LIN {X 0,Y 514.974,Z 940.438,A -85,B 0,C 180,E1 22806.113,E2 22806.113} C_VEL
LIN {X 0,Y 511.888,Z 958.496,A -85,B 0,C 180,E1 22805.05,E2 22805.05} C_VEL
LIN {X 0,Y 508.208,Z 978.384,A -85,B 0,C 180,E1 22803.67,E2 22803.67} C_VEL
LIN {X 0,Y 504.574,Z 996.273,A -85,B 0,C 180,E1 22802.202,E2 22802.202} C_VEL
LIN {X 0,Y 500.609,Z 1014.935,A -85,B 0,C 180,E1 22800.42,E2 22800.42} C_VEL
LIN {X 0,Y 500.137,Z 1017.069,A -85,B 0,C 180,E1 22800.192,E2 22800.192} C_VEL
LIN {X 0,Y 498.01,Z 1022.89,A -85,B 0,C 180,E1 22799.633,E2 22799.633} C_VEL
LIN {X 0,Y 489.476,Z 1037.041,A -85,B 0,C 180,E1 22798.306,E2 22798.306} C_VEL
LIN {X 0,Y 487.395,Z 1042.192,A -85,B 0,C 180,E1 22797.684,E2 22797.684} C_VEL
LIN {X 0,Y 483.645,Z 1058.175,A -85,B 0,C 180,E1 22795.338,E2 22795.338} C_VEL
LIN {X 0,Y 480.612,Z 1071.674,A -85,B 0,C 180,E1 22793.025,E2 22793.025} C_VEL
LIN {X 0,Y 477.995,Z 1083.738,A -85,B 0,C 180,E1 22790.575,E2 22790.575} C_VEL
LIN {X 0,Y 475.867,Z 1094.639,A -85,B 0,C 180,E1 22787.992,E2 22787.992} C_VEL
LIN {X 0,Y 474.237,Z 1103.992,A -85,B 0,C 180,E1 22785.281,E2 22785.281} C_VEL
LIN {X 0,Y 473.115,Z 1112.013,A -85,B 0,C 180,E1 22782.449,E2 22782.449} C_VEL
LIN {X 0,Y 472.494,Z 1117.73,A -85,B 0,C 180,E1 22779.87,E2 22779.87} C_VEL
LIN {X 0,Y 472.112,Z 1122.616,A -85,B 0,C 180,E1 22776.934,E2 22776.934} C_VEL
LIN {X 0,Y 471.982,Z 1125.43,A -85,B 0,C 180,E1 22774.374,E2 22774.374} C_VEL
LIN {X 0,Y 471.935,Z 1127.131,A -85,B 0,C 180,E1 22771.457,E2 22771.457} C_VEL
LIN {X 0,Y 471.943,Z 1127.212,A -85,B 0,C 180,E1 22768.907,E2 22768.907} C_VEL
LIN {X 0,Y 471.968,Z 1125.953,A -85,B 0,C 180,E1 22766.113,E2 22766.113} C_VEL
LIN {X 0,Y 472.089,Z 1123.143,A -85,B 0,C 180,E1 22763.39,E2 22763.39} C_VEL
LIN {X 0,Y 472.386,Z 1118.901,A -85,B 0,C 180,E1 22760.62,E2 22760.62} C_VEL
LIN {X 0,Y 472.973,Z 1113.117,A -85,B 0,C 180,E1 22757.919,E2 22757.919} C_VEL
LIN {X 0,Y 474.03,Z 1105.47,A -85,B 0,C 180,E1 22755.088,E2 22755.088} C_VEL
LIN {X 0,Y 475.474,Z 1096.754,A -85,B 0,C 180,E1 22752.499,E2 22752.499} C_VEL
LIN {X 0,Y 477.693,Z 1085.268,A -85,B 0,C 180,E1 22749.668,E2 22749.668} C_VEL
LIN {X 0,Y 480.112,Z 1073.916,A -85,B 0,C 180,E1 22747.31,E2 22747.31} C_VEL
LIN {X 0,Y 483.191,Z 1060.24,A -85,B 0,C 180,E1 22744.899,E2 22744.899} C_VEL
LIN {X 0,Y 486.557,Z 1045.907,A -85,B 0,C 180,E1 22742.724,E2 22742.724} C_VEL
LIN {X 0,Y 490.327,Z 1029.688,A -85,B 0,C 180,E1 22740.631,E2 22740.631} C_VEL
LIN {X 0,Y 494.255,Z 1012.751,A -85,B 0,C 180,E1 22738.738,E2 22738.738} C_VEL
LIN {X 0,Y 498.243,Z 994.544,A -85,B 0,C 180,E1 22737.02,E2 22737.02} C_VEL
LIN {X 0,Y 502.323,Z 975.012,A -85,B 0,C 180,E1 22735.437,E2 22735.437} C_VEL
LIN {X 0,Y 505.787,Z 956.671,A -85,B 0,C 180,E1 22734.185,E2 22734.185} C_VEL
LIN {X 0,Y 509.321,Z 936.541,A -85,B 0,C 180,E1 22733.014,E2 22733.014} C_VEL
LIN {X 0,Y 512.447,Z 915.409,A -85,B 0,C 180,E1 22732.011,E2 22732.011} C_VEL
LIN {X 0,Y 515.345,Z 892.845,A -85,B 0,C 180,E1 22731.144,E2 22731.144} C_VEL
LIN {X 0,Y 517.532,Z 870.869,A -85,B 0,C 180,E1 22730.501,E2 22730.501} C_VEL
LIN {X 0,Y 519.328,Z 846.322,A -85,B 0,C 180,E1 22729.983,E2 22729.983} C_VEL
LIN {X 0,Y 527.013,Z 617.451,A -85,B 0,C 180,E1 22726.684,E2 22726.684} C_VEL
LIN {X 0,Y 529.08,Z 555.866,A -85,B 0,C 180,E1 22725.782,E2 22725.782} C_VEL
LIN {X 0,Y 524.909,Z 533.069,A -85,B 0,C 180,E1 22724.874,E2 22724.874} C_VEL
LIN {X 0,Y 515.36,Z 516.714,A -85,B 0,C 180,E1 22723.399,E2 22723.399} C_VEL
LIN {X 0,Y 504.426,Z 499.31,A -85,B 0,C 180,E1 22721.61,E2 22721.61} C_VEL
LIN {X 0,Y 497.117,Z 487.981,A -85,B 0,C 180,E1 22720.29,E2 22720.29} C_VEL
LIN {X 0,Y 491.248,Z 474.305,A -85,B 0,C 180,E1 22717.635,E2 22717.635} C_VEL
LIN {X 0,Y 486.199,Z 463.352,A -85,B 0,C 180,E1 22715.269,E2 22715.269} C_VEL
LIN {X 0,Y 482.496,Z 455.619,A -85,B 0,C 180,E1 22713.452,E2 22713.452} C_VEL
LIN {X 0,Y 480.184,Z 450.949,A -85,B 0,C 180,E1 22712.283,E2 22712.283} C_VEL
LIN {X 0,Y 478.108,Z 446.81,A -85,B 0,C 180,E1 22711.2,E2 22711.2} C_VEL
LIN {X 0,Y 475.909,Z 442.427,A -85,B 0,C 180,E1 22710.003,E2 22710.003} C_VEL
LIN {X 0,Y 474.193,Z 438.99,A -85,B 0,C 180,E1 22709.011,E2 22709.011} C_VEL
LIN {X 0,Y 474.091,Z 438.231,A -85,B 0,C 180,E1 22708.672,E2 22708.672} C_VEL
LIN {X 0,Y 474.033,Z 438.161,A -85,B 0,C 180,E1 22705.086,E2 22705.086} C_VEL
LIN {X 0,Y 474.022,Z 438.165,A -85,B 0,C 180,E1 22701.663,E2 22701.663} C_VEL
LIN {X 0,Y 474.067,Z 438.17,A -85,B 0,C 180,E1 22698.189,E2 22698.189} C_VEL
LIN {X 0,Y 474.07,Z 438.181,A -85,B 0,C 180,E1 22694.661,E2 22694.661} C_VEL
LIN {X 0,Y 474.036,Z 438.17,A -85,B 0,C 180,E1 22691.19,E2 22691.19} C_VEL
LIN {X 0,Y 474.042,Z 438.155,A -85,B 0,C 180,E1 22687.514,E2 22687.514} C_VEL
LIN {X 0,Y 474.09,Z 438.146,A -85,B 0,C 180,E1 22684.112,E2 22684.112} C_VEL
LIN {X 0,Y 474.07,Z 438.166,A -85,B 0,C 180,E1 22680.604,E2 22680.604} C_VEL
LIN {X 0,Y 474.053,Z 438.18,A -85,B 0,C 180,E1 22677.098,E2 22677.098} C_VEL
LIN {X 0,Y 474.066,Z 438.161,A -85,B 0,C 180,E1 22673.46,E2 22673.46} C_VEL
LIN {X 0,Y 474.105,Z 438.145,A -85,B 0,C 180,E1 22670.034,E2 22670.034} C_VEL
LIN {X 0,Y 474.076,Z 438.152,A -85,B 0,C 180,E1 22666.461,E2 22666.461} C_VEL
LIN {X 0,Y 474.067,Z 438.164,A -85,B 0,C 180,E1 22662.952,E2 22662.952} C_VEL
LIN {X 0,Y 474.094,Z 438.17,A -85,B 0,C 180,E1 22659.377,E2 22659.377} C_VEL
LIN {X 0,Y 474.117,Z 438.173,A -85,B 0,C 180,E1 22655.849,E2 22655.849} C_VEL
LIN {X 0,Y 474.103,Z 438.234,A -85,B 0,C 180,E1 22652.219,E2 22652.219} C_VEL
LIN {X 0,Y 474.211,Z 438.738,A -85,B 0,C 180,E1 22651.884,E2 22651.884} C_VEL
LIN {X 0,Y 476.008,Z 442.457,A -85,B 0,C 180,E1 22650.834,E2 22650.834} C_VEL
LIN {X 0,Y 479.297,Z 448.858,A -85,B 0,C 180,E1 22649.123,E2 22649.123} C_VEL
LIN {X 0,Y 481.852,Z 453.929,A -85,B 0,C 180,E1 22647.849,E2 22647.849} C_VEL
LIN {X 0,Y 485.845,Z 461.926,A -85,B 0,C 180,E1 22645.959,E2 22645.959} C_VEL
LIN {X 0,Y 487.43,Z 464.88,A -85,B 0,C 180,E1 22645.373,E2 22645.373} C_VEL
LIN {X 0,Y 499.532,Z 481.118,A -85,B 0,C 180,E1 22643.148,E2 22643.148} C_VEL
LIN {X 0,Y 512.045,Z 499.258,A -85,B 0,C 180,E1 22641.039,E2 22641.039} C_VEL
LIN {X 0,Y 523.907,Z 517.752,A -85,B 0,C 180,E1 22639.181,E2 22639.181} C_VEL
LIN {X 0,Y 531.983,Z 531.498,A -85,B 0,C 180,E1 22637.975,E2 22637.975} C_VEL
LIN {X 0,Y 522.698,Z 768.418,A -85,B 0,C 180,E1 22634.376,E2 22634.376} C_VEL
LIN {X 0,Y 519.654,Z 844.715,A -85,B 0,C 180,E1 22633.19,E2 22633.19} C_VEL
LIN {X 0,Y 517.66,Z 869.839,A -85,B 0,C 180,E1 22632.628,E2 22632.628} C_VEL
LIN {X 0,Y 515.301,Z 892.72,A -85,B 0,C 180,E1 22631.945,E2 22631.945} C_VEL
LIN {X 0,Y 512.362,Z 915.91,A -85,B 0,C 180,E1 22631.048,E2 22631.048} C_VEL
LIN {X 0,Y 509.382,Z 936.467,A -85,B 0,C 180,E1 22630.08,E2 22630.08} C_VEL
LIN {X 0,Y 505.522,Z 959.82,A -85,B 0,C 180,E1 22628.757,E2 22628.757} C_VEL
LIN {X 0,Y 502.089,Z 978.916,A -85,B 0,C 180,E1 22627.474,E2 22627.474} C_VEL
LIN {X 0,Y 497.871,Z 1000.724,A -85,B 0,C 180,E1 22625.763,E2 22625.763} C_VEL
LIN {X 0,Y 494.305,Z 1018.112,A -85,B 0,C 180,E1 22624.174,E2 22624.174} C_VEL
LIN {X 0,Y 490.354,Z 1037.041,A -85,B 0,C 180,E1 22622.195,E2 22622.195} C_VEL
LIN {X 0,Y 486.762,Z 1053.913,A -85,B 0,C 180,E1 22620.139,E2 22620.139} C_VEL
LIN {X 0,Y 483.383,Z 1070.255,A -85,B 0,C 180,E1 22617.871,E2 22617.871} C_VEL
LIN {X 0,Y 480.434,Z 1084.78,A -85,B 0,C 180,E1 22615.519,E2 22615.519} C_VEL
LIN {X 0,Y 477.873,Z 1098.534,A -85,B 0,C 180,E1 22612.979,E2 22612.979} C_VEL
LIN {X 0,Y 475.763,Z 1110.817,A -85,B 0,C 180,E1 22610.29,E2 22610.29} C_VEL
LIN {X 0,Y 474.199,Z 1121.612,A -85,B 0,C 180,E1 22607.549,E2 22607.549} C_VEL
LIN {X 0,Y 473.122,Z 1130.443,A -85,B 0,C 180,E1 22604.816,E2 22604.816} C_VEL
LIN {X 0,Y 472.485,Z 1137.458,A -85,B 0,C 180,E1 22602.218,E2 22602.218} C_VEL
LIN {X 0,Y 472.088,Z 1143.705,A -85,B 0,C 180,E1 22599.249,E2 22599.249} C_VEL
LIN {X 0,Y 471.972,Z 1147.524,A -85,B 0,C 180,E1 22596.814,E2 22596.814} C_VEL
LIN {X 0,Y 471.934,Z 1150.574,A -85,B 0,C 180,E1 22594.009,E2 22594.009} C_VEL
LIN {X 0,Y 471.933,Z 1151.919,A -85,B 0,C 180,E1 22591.214,E2 22591.214} C_VEL
LIN {X 0,Y 471.93,Z 1151.942,A -85,B 0,C 180,E1 22588.907,E2 22588.907} C_VEL
LIN {X 0,Y 471.931,Z 1150.773,A -85,B 0,C 180,E1 22586.307,E2 22586.307} C_VEL
LIN {X 0,Y 471.964,Z 1147.852,A -85,B 0,C 180,E1 22583.431,E2 22583.431} C_VEL
LIN {X 0,Y 472.068,Z 1144.104,A -85,B 0,C 180,E1 22580.982,E2 22580.982} C_VEL
LIN {X 0,Y 472.41,Z 1138.385,A -85,B 0,C 180,E1 22578.152,E2 22578.152} C_VEL
LIN {X 0,Y 473.04,Z 1131.162,A -85,B 0,C 180,E1 22575.431,E2 22575.431} C_VEL
LIN {X 0,Y 473.962,Z 1123.279,A -85,B 0,C 180,E1 22572.948,E2 22572.948} C_VEL
LIN {X 0,Y 475.544,Z 1112.173,A -85,B 0,C 180,E1 22570.031,E2 22570.031} C_VEL
LIN {X 0,Y 477.369,Z 1101.223,A -85,B 0,C 180,E1 22567.591,E2 22567.591} C_VEL
LIN {X 0,Y 480.025,Z 1086.91,A -85,B 0,C 180,E1 22564.854,E2 22564.854} C_VEL
LIN {X 0,Y 482.698,Z 1073.379,A -85,B 0,C 180,E1 22562.621,E2 22562.621} C_VEL
LIN {X 0,Y 486.389,Z 1055.696,A -85,B 0,C 180,E1 22560.098,E2 22560.098} C_VEL
LIN {X 0,Y 489.701,Z 1039.918,A -85,B 0,C 180,E1 22558.147,E2 22558.147} C_VEL
LIN {X 0,Y 493.993,Z 1019.506,A -85,B 0,C 180,E1 22555.967,E2 22555.967} C_VEL
LIN {X 0,Y 497.576,Z 1001.995,A -85,B 0,C 180,E1 22554.355,E2 22554.355} C_VEL
LIN {X 0,Y 501.927,Z 979.629,A -85,B 0,C 180,E1 22552.584,E2 22552.584} C_VEL
LIN {X 0,Y 505.349,Z 960.615,A -85,B 0,C 180,E1 22551.3,E2 22551.3} C_VEL
LIN {X 0,Y 509.174,Z 937.611,A -85,B 0,C 180,E1 22549.984,E2 22549.984} C_VEL
LIN {X 0,Y 512.166,Z 917.021,A -85,B 0,C 180,E1 22549.007,E2 22549.007} C_VEL
LIN {X 0,Y 515.216,Z 893.121,A -85,B 0,C 180,E1 22548.075,E2 22548.075} C_VEL
LIN {X 0,Y 517.586,Z 870.113,A -85,B 0,C 180,E1 22547.385,E2 22547.385} C_VEL
LIN {X 0,Y 519.577,Z 845.22,A -85,B 0,C 180,E1 22546.825,E2 22546.825} C_VEL
LIN {X 0,Y 522.328,Z 776.987,A -85,B 0,C 180,E1 22545.762,E2 22545.762} C_VEL
LIN {X 0,Y 531.499,Z 541.74,A -85,B 0,C 180,E1 22542.186,E2 22542.186} C_VEL
LIN {X 0,Y 531.834,Z 531.038,A -85,B 0,C 180,E1 22542.014,E2 22542.014} C_VEL
LIN {X 0,Y 519.165,Z 510.17,A -85,B 0,C 180,E1 22540.108,E2 22540.108} C_VEL
LIN {X 0,Y 506.446,Z 491.019,A -85,B 0,C 180,E1 22538.06,E2 22538.06} C_VEL
LIN {X 0,Y 494.73,Z 474.66,A -85,B 0,C 180,E1 22536.025,E2 22536.025} C_VEL
LIN {X 0,Y 486.873,Z 464.103,A -85,B 0,C 180,E1 22534.529,E2 22534.529} C_VEL
LIN {X 0,Y 482.962,Z 456.048,A -85,B 0,C 180,E1 22532.708,E2 22532.708} C_VEL
LIN {X 0,Y 480.419,Z 451.159,A -85,B 0,C 180,E1 22531.494,E2 22531.494} C_VEL
LIN {X 0,Y 478.261,Z 446.86,A -85,B 0,C 180,E1 22530.394,E2 22530.394} C_VEL
LIN {X 0,Y 475.915,Z 442.341,A -85,B 0,C 180,E1 22529.172,E2 22529.172} C_VEL
LIN {X 0,Y 474.23,Z 438.807,A -85,B 0,C 180,E1 22528.183,E2 22528.183} C_VEL
LIN {X 0,Y 474.102,Z 438.209,A -85,B 0,C 180,E1 22527.781,E2 22527.781} C_VEL
LIN {X 0,Y 474.118,Z 438.172,A -85,B 0,C 180,E1 22524.151,E2 22524.151} C_VEL
LIN {X 0,Y 474.103,Z 438.171,A -85,B 0,C 180,E1 22520.543,E2 22520.543} C_VEL
LIN {X 0,Y 474.069,Z 438.163,A -85,B 0,C 180,E1 22517.048,E2 22517.048} C_VEL
LIN {X 0,Y 474.07,Z 438.154,A -85,B 0,C 180,E1 22513.415,E2 22513.415} C_VEL
LIN {X 0,Y 474.108,Z 438.145,A -85,B 0,C 180,E1 22509.959,E2 22509.959} C_VEL
LIN {X 0,Y 474.069,Z 438.161,A -85,B 0,C 180,E1 22506.54,E2 22506.54} C_VEL
LIN {X 0,Y 474.055,Z 438.18,A -85,B 0,C 180,E1 22502.902,E2 22502.902} C_VEL
LIN {X 0,Y 474.075,Z 438.165,A -85,B 0,C 180,E1 22499.396,E2 22499.396} C_VEL
LIN {X 0,Y 474.092,Z 438.145,A -85,B 0,C 180,E1 22495.888,E2 22495.888} C_VEL
LIN {X 0,Y 474.047,Z 438.155,A -85,B 0,C 180,E1 22492.463,E2 22492.463} C_VEL
LIN {X 0,Y 474.043,Z 438.171,A -85,B 0,C 180,E1 22488.81,E2 22488.81} C_VEL
LIN {X 0,Y 474.079,Z 438.18,A -85,B 0,C 180,E1 22485.339,E2 22485.339} C_VEL
LIN {X 0,Y 474.069,Z 438.167,A -85,B 0,C 180,E1 22481.811,E2 22481.811} C_VEL
LIN {X 0,Y 474.027,Z 438.163,A -85,B 0,C 180,E1 22478.337,E2 22478.337} C_VEL
LIN {X 0,Y 474.035,Z 438.161,A -85,B 0,C 180,E1 22474.781,E2 22474.781} C_VEL
LIN {X 0,Y 474.087,Z 438.218,A -85,B 0,C 180,E1 22471.257,E2 22471.257} C_VEL
LIN {X 0,Y 474.125,Z 438.668,A -85,B 0,C 180,E1 22470.932,E2 22470.932} C_VEL
LIN {X 0,Y 475.635,Z 442.084,A -85,B 0,C 180,E1 22469.978,E2 22469.978} C_VEL
LIN {X 0,Y 476.655,Z 443.662,A -85,B 0,C 180,E1 22469.492,E2 22469.492} C_VEL
LIN {X 0,Y 478.533,Z 447.391,A -85,B 0,C 180,E1 22468.487,E2 22468.487} C_VEL
LIN {X 0,Y 481.515,Z 453.713,A -85,B 0,C 180,E1 22466.898,E2 22466.898} C_VEL
LIN {X 0,Y 485.309,Z 461.34,A -85,B 0,C 180,E1 22465.056,E2 22465.056} C_VEL
LIN {X 0,Y 491.281,Z 474.454,A -85,B 0,C 180,E1 22462.221,E2 22462.221} C_VEL
LIN {X 0,Y 497.06,Z 487.845,A -85,B 0,C 180,E1 22459.628,E2 22459.628} C_VEL
LIN {X 0,Y 499.745,Z 492.282,A -85,B 0,C 180,E1 22459.079,E2 22459.079} C_VEL
LIN {X 0,Y 510.188,Z 508.318,A -85,B 0,C 180,E1 22457.323,E2 22457.323} C_VEL
LIN {X 0,Y 522.638,Z 529.103,A -85,B 0,C 180,E1 22455.363,E2 22455.363} C_VEL
LIN {X 0,Y 525.199,Z 534.086,A -85,B 0,C 180,E1 22454.967,E2 22454.967} C_VEL
LIN {X 0,Y 529.111,Z 557.421,A -85,B 0,C 180,E1 22454.081,E2 22454.081} C_VEL
LIN {X 0,Y 520.357,Z 817.692,A -85,B 0,C 180,E1 22450.349,E2 22450.349} C_VEL
LIN {X 0,Y 518.943,Z 852.159,A -85,B 0,C 180,E1 22449.818,E2 22449.818} C_VEL
LIN {X 0,Y 517.154,Z 874.464,A -85,B 0,C 180,E1 22449.31,E2 22449.31} C_VEL
LIN {X 0,Y 514.604,Z 898.665,A -85,B 0,C 180,E1 22448.552,E2 22448.552} C_VEL
LIN {X 0,Y 511.976,Z 918.576,A -85,B 0,C 180,E1 22447.754,E2 22447.754} C_VEL
LIN {X 0,Y 508.507,Z 941.041,A -85,B 0,C 180,E1 22446.64,E2 22446.64} C_VEL
LIN {X 0,Y 505.173,Z 959.846,A -85,B 0,C 180,E1 22445.516,E2 22445.516} C_VEL
LIN {X 0,Y 501.125,Z 980.634,A -85,B 0,C 180,E1 22444.034,E2 22444.034} C_VEL
LIN {X 0,Y 497.359,Z 998.511,A -85,B 0,C 180,E1 22442.533,E2 22442.533} C_VEL
LIN {X 0,Y 493.253,Z 1016.9,A -85,B 0,C 180,E1 22440.72,E2 22440.72} C_VEL
LIN {X 0,Y 489.571,Z 1032.936,A -85,B 0,C 180,E1 22438.883,E2 22438.883} C_VEL
LIN {X 0,Y 487.395,Z 1042.192,A -85,B 0,C 180,E1 22437.684,E2 22437.684} C_VEL
LIN {X 0,Y 485.339,Z 1047.343,A -85,B 0,C 180,E1 22437.042,E2 22437.042} C_VEL
LIN {X 0,Y 476.907,Z 1060.015,A -85,B 0,C 180,E1 22435.473,E2 22435.473} C_VEL
LIN {X 0,Y 474.868,Z 1064.523,A -85,B 0,C 180,E1 22434.753,E2 22434.753} C_VEL
LIN {X 0,Y 471.929,Z 1076.945,A -85,B 0,C 180,E1 22432.419,E2 22432.419} C_VEL
LIN {X 0,Y 469.326,Z 1088.898,A -85,B 0,C 180,E1 22429.801,E2 22429.801} C_VEL
LIN {X 0,Y 467.35,Z 1098.886,A -85,B 0,C 180,E1 22427.173,E2 22427.173} C_VEL
LIN {X 0,Y 465.767,Z 1108.276,A -85,B 0,C 180,E1 22424.166,E2 22424.166} C_VEL
LIN {X 0,Y 464.847,Z 1115.168,A -85,B 0,C 180,E1 22421.414,E2 22421.414} C_VEL
LIN {X 0,Y 464.295,Z 1120.599,A -85,B 0,C 180,E1 22418.546,E2 22418.546} C_VEL
LIN {X 0,Y 464.05,Z 1124.214,A -85,B 0,C 180,E1 22415.937,E2 22415.937} C_VEL
LIN {X 0,Y 463.959,Z 1126.617,A -85,B 0,C 180,E1 22413.089,E2 22413.089} C_VEL
LIN {X 0,Y 463.943,Z 1127.492,A -85,B 0,C 180,E1 22410.617,E2 22410.617} C_VEL
LIN {X 0,Y 463.948,Z 1127.06,A -85,B 0,C 180,E1 22407.653,E2 22407.653} C_VEL
LIN {X 0,Y 464,Z 1125.29,A -85,B 0,C 180,E1 22405.055,E2 22405.055} C_VEL
LIN {X 0,Y 464.2,Z 1121.946,A -85,B 0,C 180,E1 22402.201,E2 22402.201} C_VEL
LIN {X 0,Y 464.608,Z 1117.157,A -85,B 0,C 180,E1 22399.459,E2 22399.459} C_VEL
LIN {X 0,Y 465.431,Z 1110.588,A -85,B 0,C 180,E1 22396.584,E2 22396.584} C_VEL
LIN {X 0,Y 466.624,Z 1102.952,A -85,B 0,C 180,E1 22393.953,E2 22393.953} C_VEL
LIN {X 0,Y 468.533,Z 1092.768,A -85,B 0,C 180,E1 22391.072,E2 22391.072} C_VEL
LIN {X 0,Y 470.779,Z 1082.168,A -85,B 0,C 180,E1 22388.573,E2 22388.573} C_VEL
LIN {X 0,Y 473.781,Z 1069.027,A -85,B 0,C 180,E1 22385.963,E2 22385.963} C_VEL
LIN {X 0,Y 477.129,Z 1055.239,A -85,B 0,C 180,E1 22383.623,E2 22383.623} C_VEL
LIN {X 0,Y 480.825,Z 1039.945,A -85,B 0,C 180,E1 22381.426,E2 22381.426} C_VEL
LIN {X 0,Y 484.873,Z 1023.467,A -85,B 0,C 180,E1 22379.379,E2 22379.379} C_VEL
LIN {X 0,Y 488.838,Z 1006.54,A -85,B 0,C 180,E1 22377.594,E2 22377.594} C_VEL
LIN {X 0,Y 493.061,Z 987.865,A -85,B 0,C 180,E1 22375.894,E2 22375.894} C_VEL
LIN {X 0,Y 496.966,Z 969.009,A -85,B 0,C 180,E1 22374.446,E2 22374.446} C_VEL
LIN {X 0,Y 501.016,Z 947.927,A -85,B 0,C 180,E1 22373.079,E2 22373.079} C_VEL
LIN {X 0,Y 504.386,Z 927.99,A -85,B 0,C 180,E1 22372.009,E2 22372.009} C_VEL
LIN {X 0,Y 507.772,Z 904.722,A -85,B 0,C 180,E1 22370.991,E2 22370.991} C_VEL
LIN {X 0,Y 510.184,Z 884.575,A -85,B 0,C 180,E1 22370.295,E2 22370.295} C_VEL
LIN {X 0,Y 512.428,Z 860.395,A -85,B 0,C 180,E1 22369.663,E2 22369.663} C_VEL
LIN {X 0,Y 513.755,Z 838.487,A -85,B 0,C 180,E1 22369.26,E2 22369.26} C_VEL
LIN {X 0,Y 522.47,Z 588.071,A -85,B 0,C 180,E1 22365.635,E2 22365.635} C_VEL
LIN {X 0,Y 523.48,Z 557.529,A -85,B 0,C 180,E1 22365.174,E2 22365.174} C_VEL
LIN {X 0,Y 519.86,Z 537.391,A -85,B 0,C 180,E1 22364.359,E2 22364.359} C_VEL
LIN {X 0,Y 508.793,Z 518.402,A -85,B 0,C 180,E1 22362.592,E2 22362.592} C_VEL
LIN {X 0,Y 497.226,Z 500.156,A -85,B 0,C 180,E1 22360.62,E2 22360.62} C_VEL
LIN {X 0,Y 488.867,Z 487.482,A -85,B 0,C 180,E1 22359.047,E2 22359.047} C_VEL
LIN {X 0,Y 482.492,Z 473.005,A -85,B 0,C 180,E1 22356.054,E2 22356.054} C_VEL
LIN {X 0,Y 477.244,Z 461.72,A -85,B 0,C 180,E1 22353.437,E2 22353.437} C_VEL
LIN {X 0,Y 472.696,Z 452.61,A -85,B 0,C 180,E1 22351.073,E2 22351.073} C_VEL
LIN {X 0,Y 470.426,Z 448.145,A -85,B 0,C 180,E1 22349.826,E2 22349.826} C_VEL
LIN {X 0,Y 468.616,Z 444.219,A -85,B 0,C 180,E1 22348.722,E2 22348.722} C_VEL
LIN {X 0,Y 466.315,Z 440.328,A -85,B 0,C 180,E1 22347.453,E2 22347.453} C_VEL
LIN {X 0,Y 466.113,Z 439.268,A -85,B 0,C 180,E1 22347.051,E2 22347.051} C_VEL
LIN {X 0,Y 466.081,Z 439.159,A -85,B 0,C 180,E1 22343.518,E2 22343.518} C_VEL
LIN {X 0,Y 466.1,Z 439.151,A -85,B 0,C 180,E1 22339.943,E2 22339.943} C_VEL
LIN {X 0,Y 466.145,Z 439.138,A -85,B 0,C 180,E1 22336.448,E2 22336.448} C_VEL
LIN {X 0,Y 466.1,Z 439.144,A -85,B 0,C 180,E1 22333.018,E2 22333.018} C_VEL
LIN {X 0,Y 466.097,Z 439.154,A -85,B 0,C 180,E1 22329.383,E2 22329.383} C_VEL
LIN {X 0,Y 466.135,Z 439.167,A -85,B 0,C 180,E1 22325.91,E2 22325.91} C_VEL
LIN {X 0,Y 466.159,Z 439.15,A -85,B 0,C 180,E1 22322.213,E2 22322.213} C_VEL
LIN {X 0,Y 466.117,Z 439.138,A -85,B 0,C 180,E1 22318.771,E2 22318.771} C_VEL
LIN {X 0,Y 466.112,Z 439.142,A -85,B 0,C 180,E1 22315.201,E2 22315.201} C_VEL
LIN {X 0,Y 466.157,Z 439.157,A -85,B 0,C 180,E1 22311.737,E2 22311.737} C_VEL
LIN {X 0,Y 466.168,Z 439.163,A -85,B 0,C 180,E1 22308.117,E2 22308.117} C_VEL
LIN {X 0,Y 466.133,Z 439.151,A -85,B 0,C 180,E1 22304.574,E2 22304.574} C_VEL
LIN {X 0,Y 466.131,Z 439.143,A -85,B 0,C 180,E1 22300.971,E2 22300.971} C_VEL
LIN {X 0,Y 466.163,Z 439.137,A -85,B 0,C 180,E1 22297.422,E2 22297.422} C_VEL
LIN {X 0,Y 466.2,Z 439.306,A -85,B 0,C 180,E1 22293.704,E2 22293.704} C_VEL
LIN {X 0,Y 467.592,Z 442.857,A -85,B 0,C 180,E1 22292.629,E2 22292.629} C_VEL
LIN {X 0,Y 468.898,Z 444.787,A -85,B 0,C 180,E1 22291.986,E2 22291.986} C_VEL
LIN {X 0,Y 470.858,Z 448.554,A -85,B 0,C 180,E1 22290.903,E2 22290.903} C_VEL
LIN {X 0,Y 474.049,Z 455.088,A -85,B 0,C 180,E1 22289.166,E2 22289.166} C_VEL
LIN {X 0,Y 476.499,Z 459.914,A -85,B 0,C 180,E1 22287.934,E2 22287.934} C_VEL
LIN {X 0,Y 479.224,Z 465.188,A -85,B 0,C 180,E1 22286.719,E2 22286.719} C_VEL
LIN {X 0,Y 489.277,Z 478.497,A -85,B 0,C 180,E1 22284.738,E2 22284.738} C_VEL
LIN {X 0,Y 500.655,Z 494.217,A -85,B 0,C 180,E1 22282.689,E2 22282.689} C_VEL
LIN {X 0,Y 514.237,Z 514.73,A -85,B 0,C 180,E1 22280.428,E2 22280.428} C_VEL
LIN {X 0,Y 526.322,Z 534.731,A -85,B 0,C 180,E1 22278.555,E2 22278.555} C_VEL
LIN {X 0,Y 516.712,Z 771.522,A -85,B 0,C 180,E1 22274.93,E2 22274.93} C_VEL
LIN {X 0,Y 513.667,Z 844.882,A -85,B 0,C 180,E1 22273.779,E2 22273.779} C_VEL
LIN {X 0,Y 511.619,Z 869.914,A -85,B 0,C 180,E1 22273.215,E2 22273.215} C_VEL
LIN {X 0,Y 509.182,Z 892.812,A -85,B 0,C 180,E1 22272.526,E2 22272.526} C_VEL
LIN {X 0,Y 506.053,Z 916.585,A -85,B 0,C 180,E1 22271.597,E2 22271.597} C_VEL
LIN {X 0,Y 502.816,Z 938.112,A -85,B 0,C 180,E1 22270.567,E2 22270.567} C_VEL
LIN {X 0,Y 498.979,Z 960.274,A -85,B 0,C 180,E1 22269.289,E2 22269.289} C_VEL
LIN {X 0,Y 495.311,Z 979.929,A -85,B 0,C 180,E1 22267.949,E2 22267.949} C_VEL
LIN {X 0,Y 490.905,Z 1001.712,A -85,B 0,C 180,E1 22266.206,E2 22266.206} C_VEL
LIN {X 0,Y 487.171,Z 1019.225,A -85,B 0,C 180,E1 22264.576,E2 22264.576} C_VEL
LIN {X 0,Y 482.69,Z 1039.61,A -85,B 0,C 180,E1 22262.377,E2 22262.377} C_VEL
LIN {X 0,Y 479.163,Z 1055.625,A -85,B 0,C 180,E1 22260.372,E2 22260.372} C_VEL
LIN {X 0,Y 475.338,Z 1073.128,A -85,B 0,C 180,E1 22257.839,E2 22257.839} C_VEL
LIN {X 0,Y 472.519,Z 1086.661,A -85,B 0,C 180,E1 22255.574,E2 22255.574} C_VEL
LIN {X 0,Y 469.713,Z 1100.979,A -85,B 0,C 180,E1 22252.795,E2 22252.795} C_VEL
LIN {X 0,Y 467.841,Z 1111.624,A -85,B 0,C 180,E1 22250.388,E2 22250.388} C_VEL
LIN {X 0,Y 466.165,Z 1122.631,A -85,B 0,C 180,E1 22247.475,E2 22247.475} C_VEL
LIN {X 0,Y 465.169,Z 1130.574,A -85,B 0,C 180,E1 22244.948,E2 22244.948} C_VEL
LIN {X 0,Y 464.477,Z 1137.856,A -85,B 0,C 180,E1 22242.179,E2 22242.179} C_VEL
LIN {X 0,Y 464.093,Z 1143.674,A -85,B 0,C 180,E1 22239.299,E2 22239.299} C_VEL
LIN {X 0,Y 463.972,Z 1147.474,A -85,B 0,C 180,E1 22236.807,E2 22236.807} C_VEL
LIN {X 0,Y 463.934,Z 1150.45,A -85,B 0,C 180,E1 22233.955,E2 22233.955} C_VEL
LIN {X 0,Y 463.935,Z 1151.71,A -85,B 0,C 180,E1 22231.235,E2 22231.235} C_VEL
LIN {X 0,Y 463.933,Z 1151.733,A -85,B 0,C 180,E1 22228.889,E2 22228.889} C_VEL
LIN {X 0,Y 463.933,Z 1150.578,A -85,B 0,C 180,E1 22226.273,E2 22226.273} C_VEL
LIN {X 0,Y 463.967,Z 1147.635,A -85,B 0,C 180,E1 22223.317,E2 22223.317} C_VEL
LIN {X 0,Y 464.081,Z 1143.883,A -85,B 0,C 180,E1 22220.826,E2 22220.826} C_VEL
LIN {X 0,Y 464.451,Z 1138.157,A -85,B 0,C 180,E1 22217.946,E2 22217.946} C_VEL
LIN {X 0,Y 465.125,Z 1130.926,A -85,B 0,C 180,E1 22215.178,E2 22215.178} C_VEL
LIN {X 0,Y 466.104,Z 1123.037,A -85,B 0,C 180,E1 22212.651,E2 22212.651} C_VEL
LIN {X 0,Y 467.752,Z 1112.14,A -85,B 0,C 180,E1 22209.739,E2 22209.739} C_VEL
LIN {X 0,Y 469.602,Z 1101.551,A -85,B 0,C 180,E1 22207.332,E2 22207.332} C_VEL
LIN {X 0,Y 472.239,Z 1088.068,A -85,B 0,C 180,E1 22204.678,E2 22204.678} C_VEL
LIN {X 0,Y 475.161,Z 1073.88,A -85,B 0,C 180,E1 22202.286,E2 22202.286} C_VEL
LIN {X 0,Y 478.706,Z 1057.75,A -85,B 0,C 180,E1 22199.914,E2 22199.914} C_VEL
LIN {X 0,Y 482.334,Z 1041.104,A -85,B 0,C 180,E1 22197.807,E2 22197.807} C_VEL
LIN {X 0,Y 486.505,Z 1022.245,A -85,B 0,C 180,E1 22195.727,E2 22195.727} C_VEL
LIN {X 0,Y 490.457,Z 1003.654,A -85,B 0,C 180,E1 22193.973,E2 22193.973} C_VEL
LIN {X 0,Y 494.655,Z 983.311,A -85,B 0,C 180,E1 22192.304,E2 22192.304} C_VEL
LIN {X 0,Y 498.473,Z 962.883,A -85,B 0,C 180,E1 22190.886,E2 22190.886} C_VEL
LIN {X 0,Y 502.088,Z 942.395,A -85,B 0,C 180,E1 22189.667,E2 22189.667} C_VEL
LIN {X 0,Y 505.54,Z 919.912,A -85,B 0,C 180,E1 22188.557,E2 22188.557} C_VEL
LIN {X 0,Y 508.443,Z 898.448,A -85,B 0,C 180,E1 22187.683,E2 22187.683} C_VEL
LIN {X 0,Y 511.249,Z 873.168,A -85,B 0,C 180,E1 22186.878,E2 22186.878} C_VEL
LIN {X 0,Y 513.206,Z 850.605,A -85,B 0,C 180,E1 22186.34,E2 22186.34} C_VEL
LIN {X 0,Y 514.878,Z 817.028,A -85,B 0,C 180,E1 22185.773,E2 22185.773} C_VEL
LIN {X 0,Y 524.044,Z 587.339,A -85,B 0,C 180,E1 22182.252,E2 22182.252} C_VEL
LIN {X 0,Y 526.163,Z 534.506,A -85,B 0,C 180,E1 22181.437,E2 22181.437} C_VEL
LIN {X 0,Y 513.155,Z 513.054,A -85,B 0,C 180,E1 22179.418,E2 22179.418} C_VEL
LIN {X 0,Y 499.593,Z 492.761,A -85,B 0,C 180,E1 22177.152,E2 22177.152} C_VEL
LIN {X 0,Y 487.595,Z 476.133,A -85,B 0,C 180,E1 22174.971,E2 22174.971} C_VEL
LIN {X 0,Y 478.895,Z 464.709,A -85,B 0,C 180,E1 22173.235,E2 22173.235} C_VEL
LIN {X 0,Y 475.233,Z 457.278,A -85,B 0,C 180,E1 22171.453,E2 22171.453} C_VEL
LIN {X 0,Y 472.813,Z 452.565,A -85,B 0,C 180,E1 22170.22,E2 22170.22} C_VEL
LIN {X 0,Y 470.485,Z 448.08,A -85,B 0,C 180,E1 22168.983,E2 22168.983} C_VEL
LIN {X 0,Y 468.304,Z 443.715,A -85,B 0,C 180,E1 22167.74,E2 22167.74} C_VEL
LIN {X 0,Y 466.483,Z 440.609,A -85,B 0,C 180,E1 22166.752,E2 22166.752} C_VEL
LIN {X 0,Y 466.19,Z 439.239,A -85,B 0,C 180,E1 22166.293,E2 22166.293} C_VEL
LIN {X 0,Y 466.163,Z 439.138,A -85,B 0,C 180,E1 22162.578,E2 22162.578} C_VEL
LIN {X 0,Y 466.133,Z 439.143,A -85,B 0,C 180,E1 22159.029,E2 22159.029} C_VEL
LIN {X 0,Y 466.13,Z 439.149,A -85,B 0,C 180,E1 22155.298,E2 22155.298} C_VEL
LIN {X 0,Y 466.16,Z 439.162,A -85,B 0,C 180,E1 22151.758,E2 22151.758} C_VEL
LIN {X 0,Y 466.169,Z 439.158,A -85,B 0,C 180,E1 22148.138,E2 22148.138} C_VEL
LIN {X 0,Y 466.126,Z 439.143,A -85,B 0,C 180,E1 22144.552,E2 22144.552} C_VEL
LIN {X 0,Y 466.113,Z 439.137,A -85,B 0,C 180,E1 22140.983,E2 22140.983} C_VEL
LIN {X 0,Y 466.148,Z 439.146,A -85,B 0,C 180,E1 22137.541,E2 22137.541} C_VEL
LIN {X 0,Y 466.162,Z 439.163,A -85,B 0,C 180,E1 22133.843,E2 22133.843} C_VEL
LIN {X 0,Y 466.109,Z 439.157,A -85,B 0,C 180,E1 22130.368,E2 22130.368} C_VEL
LIN {X 0,Y 466.098,Z 439.146,A -85,B 0,C 180,E1 22126.73,E2 22126.73} C_VEL
LIN {X 0,Y 466.134,Z 439.139,A -85,B 0,C 180,E1 22123.295,E2 22123.295} C_VEL
LIN {X 0,Y 466.139,Z 439.142,A -85,B 0,C 180,E1 22119.666,E2 22119.666} C_VEL
LIN {X 0,Y 466.09,Z 439.154,A -85,B 0,C 180,E1 22116.214,E2 22116.214} C_VEL
LIN {X 0,Y 466.118,Z 439.345,A -85,B 0,C 180,E1 22112.705,E2 22112.705} C_VEL
LIN {X 0,Y 467.519,Z 442.769,A -85,B 0,C 180,E1 22111.654,E2 22111.654} C_VEL
LIN {X 0,Y 468.773,Z 444.831,A -85,B 0,C 180,E1 22110.99,E2 22110.99} C_VEL
LIN {X 0,Y 470.716,Z 448.486,A -85,B 0,C 180,E1 22109.913,E2 22109.913} C_VEL
LIN {X 0,Y 474.066,Z 455.517,A -85,B 0,C 180,E1 22108.035,E2 22108.035} C_VEL
LIN {X 0,Y 475.982,Z 459.387,A -85,B 0,C 180,E1 22107.038,E2 22107.038} C_VEL
LIN {X 0,Y 479.724,Z 467.049,A -85,B 0,C 180,E1 22105.173,E2 22105.173} C_VEL
LIN {X 0,Y 485.925,Z 480.762,A -85,B 0,C 180,E1 22102.179,E2 22102.179} C_VEL
LIN {X 0,Y 489.36,Z 488.411,A -85,B 0,C 180,E1 22100.698,E2 22100.698} C_VEL
LIN {X 0,Y 502.784,Z 508.809,A -85,B 0,C 180,E1 22098.3,E2 22098.3} C_VEL
LIN {X 0,Y 513.543,Z 526.486,A -85,B 0,C 180,E1 22096.525,E2 22096.525} C_VEL
LIN {X 0,Y 520.096,Z 538.242,A -85,B 0,C 180,E1 22095.489,E2 22095.489} C_VEL
LIN {X 0,Y 523.504,Z 559.063,A -85,B 0,C 180,E1 22094.688,E2 22094.688} C_VEL
LIN {X 0,Y 514.417,Z 818.312,A -85,B 0,C 180,E1 22090.939,E2 22090.939} C_VEL
LIN {X 0,Y 512.95,Z 852.446,A -85,B 0,C 180,E1 22090.406,E2 22090.406} C_VEL
LIN {X 0,Y 511.115,Z 874.559,A -85,B 0,C 180,E1 22089.898,E2 22089.898} C_VEL
LIN {X 0,Y 508.489,Z 898.644,A -85,B 0,C 180,E1 22089.14,E2 22089.14} C_VEL
LIN {X 0,Y 505.764,Z 918.625,A -85,B 0,C 180,E1 22088.333,E2 22088.333} C_VEL
LIN {X 0,Y 502.1,Z 941.54,A -85,B 0,C 180,E1 22087.186,E2 22087.186} C_VEL
LIN {X 0,Y 498.658,Z 960.303,A -85,B 0,C 180,E1 22086.052,E2 22086.052} C_VEL
LIN {X 0,Y 494.466,Z 981.024,A -85,B 0,C 180,E1 22084.557,E2 22084.557} C_VEL
LIN {X 0,Y 490.565,Z 998.877,A -85,B 0,C 180,E1 22083.041,E2 22083.041} C_VEL
LIN {X 0,Y 486.266,Z 1017.348,A -85,B 0,C 180,E1 22081.195,E2 22081.195} C_VEL
LIN {X 0,Y 482.355,Z 1033.745,A -85,B 0,C 180,E1 22079.289,E2 22079.289} C_VEL
LIN {X 0,Y 478.409,Z 1049.719,A -85,B 0,C 180,E1 22077.105,E2 22077.105} C_VEL
LIN {X 0,Y 474.895,Z 1064.42,A -85,B 0,C 180,E1 22074.771,E2 22074.771} C_VEL
LIN {X 0,Y 474.868,Z 1064.523,A -85,B 0,C 180,E1 22074.753,E2 22074.753} C_VEL
LIN {X 0,Y 472.869,Z 1068.934,A -85,B 0,C 180,E1 22074.014,E2 22074.014} C_VEL
LIN {X 0,Y 464.347,Z 1080.474,A -85,B 0,C 180,E1 22072.094,E2 22072.094} C_VEL
LIN {X 0,Y 462.869,Z 1083.71,A -85,B 0,C 180,E1 22071.406,E2 22071.406} C_VEL
LIN {X 0,Y 460.491,Z 1094.645,A -85,B 0,C 180,E1 22068.745,E2 22068.745} C_VEL
LIN {X 0,Y 458.637,Z 1104.068,A -85,B 0,C 180,E1 22065.944,E2 22065.944} C_VEL
LIN {X 0,Y 457.384,Z 1111.878,A -85,B 0,C 180,E1 22063.141,E2 22063.141} C_VEL
LIN {X 0,Y 456.602,Z 1117.927,A -85,B 0,C 180,E1 22060.345,E2 22060.345} C_VEL
LIN {X 0,Y 456.181,Z 1122.739,A -85,B 0,C 180,E1 22057.43,E2 22057.43} C_VEL
LIN {X 0,Y 455.998,Z 1125.745,A -85,B 0,C 180,E1 22054.654,E2 22054.654} C_VEL
LIN {X 0,Y 455.945,Z 1127.507,A -85,B 0,C 180,E1 22051.759,E2 22051.759} C_VEL
LIN {X 0,Y 455.945,Z 1127.675,A -85,B 0,C 180,E1 22049.12,E2 22049.12} C_VEL
LIN {X 0,Y 455.968,Z 1126.683,A -85,B 0,C 180,E1 22046.48,E2 22046.48} C_VEL
LIN {X 0,Y 456.1,Z 1123.931,A -85,B 0,C 180,E1 22043.454,E2 22043.454} C_VEL
LIN {X 0,Y 456.381,Z 1120.171,A -85,B 0,C 180,E1 22040.797,E2 22040.797} C_VEL
LIN {X 0,Y 457.021,Z 1114.441,A -85,B 0,C 180,E1 22037.876,E2 22037.876} C_VEL
LIN {X 0,Y 458.026,Z 1107.737,A -85,B 0,C 180,E1 22035.202,E2 22035.202} C_VEL
LIN {X 0,Y 459.685,Z 1098.562,A -85,B 0,C 180,E1 22032.27,E2 22032.27} C_VEL
LIN {X 0,Y 461.824,Z 1088.505,A -85,B 0,C 180,E1 22029.599,E2 22029.599} C_VEL
LIN {X 0,Y 464.447,Z 1077.034,A -85,B 0,C 180,E1 22027.066,E2 22027.066} C_VEL
LIN {X 0,Y 467.746,Z 1063.79,A -85,B 0,C 180,E1 22024.553,E2 22024.553} C_VEL
LIN {X 0,Y 471.257,Z 1049.774,A -85,B 0,C 180,E1 22022.311,E2 22022.311} C_VEL
LIN {X 0,Y 475.376,Z 1033.773,A -85,B 0,C 180,E1 22020.099,E2 22020.099} C_VEL
LIN {X 0,Y 479.359,Z 1017.737,A -85,B 0,C 180,E1 22018.212,E2 22018.212} C_VEL
LIN {X 0,Y 483.785,Z 999.521,A -85,B 0,C 180,E1 22016.364,E2 22016.364} C_VEL
LIN {X 0,Y 487.825,Z 981.716,A -85,B 0,C 180,E1 22014.833,E2 22014.833} C_VEL
LIN {X 0,Y 492.162,Z 961.118,A -85,B 0,C 180,E1 22013.323,E2 22013.323} C_VEL
LIN {X 0,Y 495.716,Z 942.431,A -85,B 0,C 180,E1 22012.179,E2 22012.179} C_VEL
LIN {X 0,Y 499.422,Z 920.323,A -85,B 0,C 180,E1 22011.049,E2 22011.049} C_VEL
LIN {X 0,Y 502.326,Z 899.813,A -85,B 0,C 180,E1 22010.206,E2 22010.206} C_VEL
LIN {X 0,Y 505.099,Z 875.664,A -85,B 0,C 180,E1 22009.429,E2 22009.429} C_VEL
LIN {X 0,Y 506.979,Z 853.897,A -85,B 0,C 180,E1 22008.918,E2 22008.918} C_VEL
LIN {X 0,Y 508.477,Z 822.337,A -85,B 0,C 180,E1 22008.41,E2 22008.41} C_VEL
LIN {X 0,Y 518.024,Z 561.104,A -85,B 0,C 180,E1 22004.601,E2 22004.601} C_VEL
LIN {X 0,Y 517.363,Z 555.729,A -85,B 0,C 180,E1 22004.417,E2 22004.417} C_VEL
LIN {X 0,Y 514.791,Z 541.58,A -85,B 0,C 180,E1 22003.824,E2 22003.824} C_VEL
LIN {X 0,Y 503.008,Z 521.469,A -85,B 0,C 180,E1 22001.887,E2 22001.887} C_VEL
LIN {X 0,Y 492.958,Z 505.545,A -85,B 0,C 180,E1 22000.12,E2 22000.12} C_VEL
LIN {X 0,Y 483.247,Z 491.186,A -85,B 0,C 180,E1 21998.294,E2 21998.294} C_VEL
LIN {X 0,Y 480.559,Z 486.973,A -85,B 0,C 180,E1 21997.714,E2 21997.714} C_VEL
LIN {X 0,Y 474.86,Z 474.299,A -85,B 0,C 180,E1 21994.942,E2 21994.942} C_VEL
LIN {X 0,Y 471.127,Z 466.43,A -85,B 0,C 180,E1 21993.036,E2 21993.036} C_VEL
LIN {X 0,Y 467.476,Z 458.681,A -85,B 0,C 180,E1 21991.03,E2 21991.03} C_VEL
LIN {X 0,Y 464.955,Z 453.849,A -85,B 0,C 180,E1 21989.645,E2 21989.645} C_VEL
LIN {X 0,Y 462.592,Z 449.185,A -85,B 0,C 180,E1 21988.253,E2 21988.253} C_VEL
LIN {X 0,Y 460.781,Z 445.498,A -85,B 0,C 180,E1 21987.11,E2 21987.11} C_VEL
LIN {X 0,Y 458.329,Z 441.147,A -85,B 0,C 180,E1 21985.592,E2 21985.592} C_VEL
LIN {X 0,Y 458.16,Z 440.226,A -85,B 0,C 180,E1 21985.187,E2 21985.187} C_VEL
LIN {X 0,Y 458.144,Z 440.14,A -85,B 0,C 180,E1 21981.606,E2 21981.606} C_VEL
LIN {X 0,Y 458.175,Z 440.144,A -85,B 0,C 180,E1 21978.053,E2 21978.053} C_VEL
LIN {X 0,Y 458.223,Z 440.151,A -85,B 0,C 180,E1 21974.404,E2 21974.404} C_VEL
LIN {X 0,Y 458.188,Z 440.154,A -85,B 0,C 180,E1 21970.69,E2 21970.69} C_VEL
LIN {X 0,Y 458.16,Z 440.136,A -85,B 0,C 180,E1 21967.146,E2 21967.146} C_VEL
LIN {X 0,Y 458.169,Z 440.126,A -85,B 0,C 180,E1 21963.503,E2 21963.503} C_VEL
LIN {X 0,Y 458.22,Z 440.126,A -85,B 0,C 180,E1 21960,E2 21960} C_VEL
LIN {X 0,Y 458.209,Z 440.149,A -85,B 0,C 180,E1 21956.372,E2 21956.372} C_VEL
LIN {X 0,Y 458.18,Z 440.152,A -85,B 0,C 180,E1 21952.854,E2 21952.854} C_VEL
LIN {X 0,Y 458.183,Z 440.135,A -85,B 0,C 180,E1 21949.124,E2 21949.124} C_VEL
LIN {X 0,Y 458.217,Z 440.123,A -85,B 0,C 180,E1 21945.596,E2 21945.596} C_VEL
LIN {X 0,Y 458.232,Z 440.121,A -85,B 0,C 180,E1 21941.95,E2 21941.95} C_VEL
LIN {X 0,Y 458.207,Z 440.128,A -85,B 0,C 180,E1 21938.359,E2 21938.359} C_VEL
LIN {X 0,Y 458.267,Z 440.4,A -85,B 0,C 180,E1 21935.485,E2 21935.485} C_VEL
LIN {X 0,Y 459.701,Z 443.884,A -85,B 0,C 180,E1 21934.352,E2 21934.352} C_VEL
LIN {X 0,Y 460.92,Z 445.502,A -85,B 0,C 180,E1 21933.734,E2 21933.734} C_VEL
LIN {X 0,Y 462.718,Z 449.291,A -85,B 0,C 180,E1 21932.595,E2 21932.595} C_VEL
LIN {X 0,Y 463.648,Z 450.851,A -85,B 0,C 180,E1 21932.097,E2 21932.097} C_VEL
LIN {X 0,Y 466.426,Z 456.493,A -85,B 0,C 180,E1 21930.5,E2 21930.5} C_VEL
LIN {X 0,Y 468.679,Z 460.964,A -85,B 0,C 180,E1 21929.291,E2 21929.291} C_VEL
LIN {X 0,Y 471.025,Z 465.441,A -85,B 0,C 180,E1 21928.162,E2 21928.162} C_VEL
LIN {X 0,Y 482.045,Z 479.809,A -85,B 0,C 180,E1 21925.857,E2 21925.857} C_VEL
LIN {X 0,Y 492.957,Z 494.785,A -85,B 0,C 180,E1 21923.789,E2 21923.789} C_VEL
LIN {X 0,Y 504.554,Z 511.949,A -85,B 0,C 180,E1 21921.754,E2 21921.754} C_VEL
LIN {X 0,Y 515.984,Z 530.201,A -85,B 0,C 180,E1 21919.884,E2 21919.884} C_VEL
LIN {X 0,Y 520.698,Z 538.411,A -85,B 0,C 180,E1 21919.142,E2 21919.142} C_VEL
LIN {X 0,Y 510.79,Z 774.183,A -85,B 0,C 180,E1 21915.505,E2 21915.505} C_VEL
LIN {X 0,Y 507.743,Z 844.957,A -85,B 0,C 180,E1 21914.384,E2 21914.384} C_VEL
LIN {X 0,Y 505.64,Z 869.933,A -85,B 0,C 180,E1 21913.818,E2 21913.818} C_VEL
LIN {X 0,Y 503.139,Z 892.716,A -85,B 0,C 180,E1 21913.128,E2 21913.128} C_VEL
LIN {X 0,Y 499.986,Z 915.973,A -85,B 0,C 180,E1 21912.218,E2 21912.218} C_VEL
LIN {X 0,Y 496.62,Z 937.647,A -85,B 0,C 180,E1 21911.177,E2 21911.177} C_VEL
LIN {X 0,Y 492.481,Z 960.733,A -85,B 0,C 180,E1 21909.834,E2 21909.834} C_VEL
LIN {X 0,Y 488.646,Z 980.541,A -85,B 0,C 180,E1 21908.467,E2 21908.467} C_VEL
LIN {X 0,Y 484.193,Z 1001.703,A -85,B 0,C 180,E1 21906.75,E2 21906.75} C_VEL
LIN {X 0,Y 480.248,Z 1019.498,A -85,B 0,C 180,E1 21905.075,E2 21905.075} C_VEL
LIN {X 0,Y 475.585,Z 1039.813,A -85,B 0,C 180,E1 21902.849,E2 21902.849} C_VEL
LIN {X 0,Y 471.945,Z 1055.604,A -85,B 0,C 180,E1 21900.845,E2 21900.845} C_VEL
LIN {X 0,Y 468.009,Z 1072.848,A -85,B 0,C 180,E1 21898.314,E2 21898.314} C_VEL
LIN {X 0,Y 465.017,Z 1086.483,A -85,B 0,C 180,E1 21896,E2 21896} C_VEL
LIN {X 0,Y 462.082,Z 1100.723,A -85,B 0,C 180,E1 21893.193,E2 21893.193} C_VEL
LIN {X 0,Y 460.101,Z 1111.374,A -85,B 0,C 180,E1 21890.746,E2 21890.746} C_VEL
LIN {X 0,Y 458.323,Z 1122.393,A -85,B 0,C 180,E1 21887.784,E2 21887.784} C_VEL
LIN {X 0,Y 457.262,Z 1130.341,A -85,B 0,C 180,E1 21885.213,E2 21885.213} C_VEL
LIN {X 0,Y 456.515,Z 1137.742,A -85,B 0,C 180,E1 21882.349,E2 21882.349} C_VEL
LIN {X 0,Y 456.108,Z 1143.523,A -85,B 0,C 180,E1 21879.423,E2 21879.423} C_VEL
LIN {X 0,Y 455.979,Z 1147.259,A -85,B 0,C 180,E1 21876.927,E2 21876.927} C_VEL
LIN {X 0,Y 455.937,Z 1150.239,A -85,B 0,C 180,E1 21874.024,E2 21874.024} C_VEL
LIN {X 0,Y 455.938,Z 1151.5,A -85,B 0,C 180,E1 21871.257,E2 21871.257} C_VEL
LIN {X 0,Y 455.936,Z 1151.523,A -85,B 0,C 180,E1 21868.869,E2 21868.869} C_VEL
LIN {X 0,Y 455.934,Z 1150.379,A -85,B 0,C 180,E1 21866.228,E2 21866.228} C_VEL
LIN {X 0,Y 455.972,Z 1147.419,A -85,B 0,C 180,E1 21863.199,E2 21863.199} C_VEL
LIN {X 0,Y 456.097,Z 1143.663,A -85,B 0,C 180,E1 21860.664,E2 21860.664} C_VEL
LIN {X 0,Y 456.497,Z 1137.93,A -85,B 0,C 180,E1 21857.733,E2 21857.733} C_VEL
LIN {X 0,Y 457.217,Z 1130.692,A -85,B 0,C 180,E1 21854.916,E2 21854.916} C_VEL
LIN {X 0,Y 458.257,Z 1122.796,A -85,B 0,C 180,E1 21852.345,E2 21852.345} C_VEL
LIN {X 0,Y 460.01,Z 1111.887,A -85,B 0,C 180,E1 21849.382,E2 21849.382} C_VEL
LIN {X 0,Y 461.992,Z 1101.136,A -85,B 0,C 180,E1 21846.902,E2 21846.902} C_VEL
LIN {X 0,Y 464.887,Z 1087.073,A -85,B 0,C 180,E1 21844.112,E2 21844.112} C_VEL
LIN {X 0,Y 467.821,Z 1073.595,A -85,B 0,C 180,E1 21841.813,E2 21841.813} C_VEL
LIN {X 0,Y 471.633,Z 1056.969,A -85,B 0,C 180,E1 21839.344,E2 21839.344} C_VEL
LIN {X 0,Y 475.332,Z 1040.784,A -85,B 0,C 180,E1 21837.274,E2 21837.274} C_VEL
LIN {X 0,Y 479.693,Z 1021.891,A -85,B 0,C 180,E1 21835.17,E2 21835.17} C_VEL
LIN {X 0,Y 483.807,Z 1003.281,A -85,B 0,C 180,E1 21833.398,E2 21833.398} C_VEL
LIN {X 0,Y 488.162,Z 982.881,A -85,B 0,C 180,E1 21831.713,E2 21831.713} C_VEL
LIN {X 0,Y 492.084,Z 962.643,A -85,B 0,C 180,E1 21830.297,E2 21830.297} C_VEL
LIN {X 0,Y 496.063,Z 940.867,A -85,B 0,C 180,E1 21828.997,E2 21828.997} C_VEL
LIN {X 0,Y 499.583,Z 918.347,A -85,B 0,C 180,E1 21827.895,E2 21827.895} C_VEL
LIN {X 0,Y 502.824,Z 895,A -85,B 0,C 180,E1 21826.955,E2 21826.955} C_VEL
LIN {X 0,Y 505.476,Z 870.97,A -85,B 0,C 180,E1 21826.217,E2 21826.217} C_VEL
LIN {X 0,Y 507.605,Z 846.421,A -85,B 0,C 180,E1 21825.648,E2 21825.648} C_VEL
LIN {X 0,Y 510.132,Z 788.884,A -85,B 0,C 180,E1 21824.73,E2 21824.73} C_VEL
LIN {X 0,Y 519.708,Z 559.361,A -85,B 0,C 180,E1 21821.185,E2 21821.185} C_VEL
LIN {X 0,Y 520.475,Z 537.838,A -85,B 0,C 180,E1 21820.836,E2 21820.836} C_VEL
LIN {X 0,Y 507.914,Z 517.177,A -85,B 0,C 180,E1 21818.83,E2 21818.83} C_VEL
LIN {X 0,Y 494.888,Z 497.553,A -85,B 0,C 180,E1 21816.586,E2 21816.586} C_VEL
LIN {X 0,Y 483.704,Z 482.039,A -85,B 0,C 180,E1 21814.5,E2 21814.5} C_VEL
LIN {X 0,Y 473.022,Z 468.109,A -85,B 0,C 180,E1 21812.331,E2 21812.331} C_VEL
LIN {X 0,Y 470.786,Z 464.994,A -85,B 0,C 180,E1 21811.784,E2 21811.784} C_VEL
LIN {X 0,Y 467.372,Z 458.269,A -85,B 0,C 180,E1 21810.041,E2 21810.041} C_VEL
LIN {X 0,Y 465.062,Z 453.804,A -85,B 0,C 180,E1 21808.79,E2 21808.79} C_VEL
LIN {X 0,Y 462.887,Z 449.487,A -85,B 0,C 180,E1 21807.534,E2 21807.534} C_VEL
LIN {X 0,Y 460.985,Z 445.752,A -85,B 0,C 180,E1 21806.387,E2 21806.387} C_VEL
LIN {X 0,Y 458.442,Z 441.289,A -85,B 0,C 180,E1 21804.861,E2 21804.861} C_VEL
LIN {X 0,Y 458.252,Z 440.278,A -85,B 0,C 180,E1 21804.493,E2 21804.493} C_VEL
LIN {X 0,Y 458.202,Z 440.14,A -85,B 0,C 180,E1 21800.935,E2 21800.935} C_VEL
LIN {X 0,Y 458.193,Z 440.134,A -85,B 0,C 180,E1 21797.265,E2 21797.265} C_VEL
LIN {X 0,Y 458.217,Z 440.124,A -85,B 0,C 180,E1 21793.76,E2 21793.76} C_VEL
LIN {X 0,Y 458.223,Z 440.122,A -85,B 0,C 180,E1 21790.181,E2 21790.181} C_VEL
LIN {X 0,Y 458.187,Z 440.139,A -85,B 0,C 180,E1 21786.642,E2 21786.642} C_VEL
LIN {X 0,Y 458.18,Z 440.159,A -85,B 0,C 180,E1 21783.002,E2 21783.002} C_VEL
LIN {X 0,Y 458.196,Z 440.141,A -85,B 0,C 180,E1 21779.375,E2 21779.375} C_VEL
LIN {X 0,Y 458.217,Z 440.122,A -85,B 0,C 180,E1 21775.742,E2 21775.742} C_VEL
LIN {X 0,Y 458.182,Z 440.126,A -85,B 0,C 180,E1 21772.21,E2 21772.21} C_VEL
LIN {X 0,Y 458.164,Z 440.143,A -85,B 0,C 180,E1 21768.673,E2 21768.673} C_VEL
LIN {X 0,Y 458.179,Z 440.158,A -85,B 0,C 180,E1 21765.077,E2 21765.077} C_VEL
LIN {X 0,Y 458.209,Z 440.147,A -85,B 0,C 180,E1 21761.554,E2 21761.554} C_VEL
LIN {X 0,Y 458.17,Z 440.143,A -85,B 0,C 180,E1 21757.953,E2 21757.953} C_VEL
LIN {X 0,Y 458.174,Z 440.326,A -85,B 0,C 180,E1 21754.537,E2 21754.537} C_VEL
LIN {X 0,Y 459.609,Z 443.783,A -85,B 0,C 180,E1 21753.374,E2 21753.374} C_VEL
LIN {X 0,Y 460.918,Z 445.955,A -85,B 0,C 180,E1 21752.619,E2 21752.619} C_VEL
LIN {X 0,Y 462.863,Z 449.485,A -85,B 0,C 180,E1 21751.483,E2 21751.483} C_VEL
LIN {X 0,Y 465.23,Z 454.206,A -85,B 0,C 180,E1 21750.091,E2 21750.091} C_VEL
LIN {X 0,Y 470.033,Z 463.983,A -85,B 0,C 180,E1 21747.439,E2 21747.439} C_VEL
LIN {X 0,Y 475.697,Z 475.944,A -85,B 0,C 180,E1 21744.54,E2 21744.54} C_VEL
LIN {X 0,Y 480.905,Z 487.753,A -85,B 0,C 180,E1 21742.054,E2 21742.054} C_VEL
LIN {X 0,Y 490.674,Z 502.13,A -85,B 0,C 180,E1 21740.18,E2 21740.18} C_VEL
LIN {X 0,Y 501.965,Z 519.774,A -85,B 0,C 180,E1 21738.179,E2 21738.179} C_VEL
LIN {X 0,Y 514.45,Z 541.07,A -85,B 0,C 180,E1 21736.12,E2 21736.12} C_VEL
LIN {X 0,Y 515.185,Z 543.242,A -85,B 0,C 180,E1 21735.987,E2 21735.987} C_VEL
LIN {X 0,Y 517.955,Z 560.731,A -85,B 0,C 180,E1 21735.308,E2 21735.308} C_VEL
LIN {X 0,Y 508.511,Z 819.577,A -85,B 0,C 180,E1 21731.533,E2 21731.533} C_VEL
LIN {X 0,Y 507.011,Z 852.726,A -85,B 0,C 180,E1 21731.008,E2 21731.008} C_VEL
LIN {X 0,Y 505.121,Z 874.759,A -85,B 0,C 180,E1 21730.497,E2 21730.497} C_VEL
LIN {X 0,Y 502.333,Z 899.354,A -85,B 0,C 180,E1 21729.714,E2 21729.714} C_VEL
LIN {X 0,Y 499.425,Z 919.947,A -85,B 0,C 180,E1 21728.87,E2 21728.87} C_VEL
LIN {X 0,Y 495.788,Z 941.772,A -85,B 0,C 180,E1 21727.76,E2 21727.76} C_VEL
LIN {X 0,Y 492.186,Z 960.755,A -85,B 0,C 180,E1 21726.602,E2 21726.602} C_VEL
LIN {X 0,Y 487.85,Z 981.409,A -85,B 0,C 180,E1 21725.093,E2 21725.093} C_VEL
LIN {X 0,Y 483.811,Z 999.239,A -85,B 0,C 180,E1 21723.562,E2 21723.562} C_VEL
LIN {X 0,Y 479.375,Z 1017.549,A -85,B 0,C 180,E1 21721.711,E2 21721.711} C_VEL
LIN {X 0,Y 475.281,Z 1034.053,A -85,B 0,C 180,E1 21719.768,E2 21719.768} C_VEL
LIN {X 0,Y 471.173,Z 1050.002,A -85,B 0,C 180,E1 21717.557,E2 21717.557} C_VEL
LIN {X 0,Y 467.5,Z 1064.684,A -85,B 0,C 180,E1 21715.19,E2 21715.19} C_VEL
LIN {X 0,Y 464.394,Z 1077.202,A -85,B 0,C 180,E1 21712.803,E2 21712.803} C_VEL
LIN {X 0,Y 462.869,Z 1083.71,A -85,B 0,C 180,E1 21711.406,E2 21711.406} C_VEL
LIN {X 0,Y 461.071,Z 1087.544,A -85,B 0,C 180,E1 21710.59,E2 21710.59} C_VEL
LIN {X 0,Y 453.012,Z 1097.021,A -85,B 0,C 180,E1 21708.432,E2 21708.432} C_VEL
LIN {X 0,Y 451.739,Z 1099.709,A -85,B 0,C 180,E1 21707.682,E2 21707.682} C_VEL
LIN {X 0,Y 450.03,Z 1108.732,A -85,B 0,C 180,E1 21704.672,E2 21704.672} C_VEL
LIN {X 0,Y 448.986,Z 1115.616,A -85,B 0,C 180,E1 21701.823,E2 21701.823} C_VEL
LIN {X 0,Y 448.367,Z 1121.033,A -85,B 0,C 180,E1 21698.852,E2 21698.852} C_VEL
LIN {X 0,Y 448.069,Z 1124.797,A -85,B 0,C 180,E1 21696.02,E2 21696.02} C_VEL
LIN {X 0,Y 447.966,Z 1127.104,A -85,B 0,C 180,E1 21693.071,E2 21693.071} C_VEL
LIN {X 0,Y 447.947,Z 1127.956,A -85,B 0,C 180,E1 21690.384,E2 21690.384} C_VEL
LIN {X 0,Y 447.955,Z 1127.35,A -85,B 0,C 180,E1 21687.313,E2 21687.313} C_VEL
LIN {X 0,Y 448.027,Z 1125.604,A -85,B 0,C 180,E1 21684.75,E2 21684.75} C_VEL
LIN {X 0,Y 448.27,Z 1121.979,A -85,B 0,C 180,E1 21681.663,E2 21681.663} C_VEL
LIN {X 0,Y 448.752,Z 1117.349,A -85,B 0,C 180,E1 21678.953,E2 21678.953} C_VEL
LIN {X 0,Y 449.766,Z 1110.355,A -85,B 0,C 180,E1 21675.845,E2 21675.845} C_VEL
LIN {X 0,Y 451.16,Z 1102.626,A -85,B 0,C 180,E1 21673.122,E2 21673.122} C_VEL
LIN {X 0,Y 453.233,Z 1092.748,A -85,B 0,C 180,E1 21670.273,E2 21670.273} C_VEL
LIN {X 0,Y 455.76,Z 1082.1,A -85,B 0,C 180,E1 21667.694,E2 21667.694} C_VEL
LIN {X 0,Y 458.919,Z 1069.545,A -85,B 0,C 180,E1 21665.133,E2 21665.133} C_VEL
LIN {X 0,Y 462.363,Z 1056.524,A -85,B 0,C 180,E1 21662.851,E2 21662.851} C_VEL
LIN {X 0,Y 466.355,Z 1041.426,A -85,B 0,C 180,E1 21660.594,E2 21660.594} C_VEL
LIN {X 0,Y 470.584,Z 1025.543,A -85,B 0,C 180,E1 21658.548,E2 21658.548} C_VEL
LIN {X 0,Y 475.092,Z 1007.799,A -85,B 0,C 180,E1 21656.608,E2 21656.608} C_VEL
LIN {X 0,Y 479.62,Z 989.329,A -85,B 0,C 180,E1 21654.873,E2 21654.873} C_VEL
LIN {X 0,Y 483.962,Z 969.812,A -85,B 0,C 180,E1 21653.338,E2 21653.338} C_VEL
LIN {X 0,Y 488.199,Z 949.4,A -85,B 0,C 180,E1 21651.978,E2 21651.978} C_VEL
LIN {X 0,Y 491.876,Z 929.052,A -85,B 0,C 180,E1 21650.862,E2 21650.862} C_VEL
LIN {X 0,Y 495.41,Z 906.648,A -85,B 0,C 180,E1 21649.852,E2 21649.852} C_VEL
LIN {X 0,Y 498.072,Z 885.927,A -85,B 0,C 180,E1 21649.117,E2 21649.117} C_VEL
LIN {X 0,Y 500.45,Z 862.678,A -85,B 0,C 180,E1 21648.484,E2 21648.484} C_VEL
LIN {X 0,Y 501.934,Z 840.461,A -85,B 0,C 180,E1 21648.058,E2 21648.058} C_VEL
LIN {X 0,Y 511.348,Z 591.684,A -85,B 0,C 180,E1 21644.392,E2 21644.392} C_VEL
LIN {X 0,Y 512.478,Z 561.029,A -85,B 0,C 180,E1 21643.925,E2 21643.925} C_VEL
LIN {X 0,Y 509.832,Z 545.97,A -85,B 0,C 180,E1 21643.29,E2 21643.29} C_VEL
LIN {X 0,Y 497.518,Z 524.776,A -85,B 0,C 180,E1 21641.201,E2 21641.201} C_VEL
LIN {X 0,Y 485.465,Z 505.877,A -85,B 0,C 180,E1 21638.993,E2 21638.993} C_VEL
LIN {X 0,Y 475.731,Z 491.689,A -85,B 0,C 180,E1 21637.063,E2 21637.063} C_VEL
LIN {X 0,Y 471.95,Z 485.935,A -85,B 0,C 180,E1 21636.176,E2 21636.176} C_VEL
LIN {X 0,Y 466.984,Z 474.871,A -85,B 0,C 180,E1 21633.6,E2 21633.6} C_VEL
LIN {X 0,Y 461.988,Z 464.365,A -85,B 0,C 180,E1 21630.86,E2 21630.86} C_VEL
LIN {X 0,Y 459.493,Z 459.543,A -85,B 0,C 180,E1 21629.459,E2 21629.459} C_VEL
LIN {X 0,Y 457.407,Z 455.245,A -85,B 0,C 180,E1 21628.176,E2 21628.176} C_VEL
LIN {X 0,Y 455.414,Z 451.168,A -85,B 0,C 180,E1 21626.891,E2 21626.891} C_VEL
LIN {X 0,Y 453.129,Z 447.241,A -85,B 0,C 180,E1 21625.486,E2 21625.486} C_VEL
LIN {X 0,Y 452.186,Z 445.445,A -85,B 0,C 180,E1 21624.843,E2 21624.843} C_VEL
LIN {X 0,Y 450.346,Z 441.94,A -85,B 0,C 180,E1 21623.512,E2 21623.512} C_VEL
LIN {X 0,Y 450.229,Z 441.237,A -85,B 0,C 180,E1 21623.147,E2 21623.147} C_VEL
LIN {X 0,Y 450.211,Z 441.137,A -85,B 0,C 180,E1 21619.46,E2 21619.46} C_VEL
LIN {X 0,Y 450.226,Z 441.126,A -85,B 0,C 180,E1 21615.853,E2 21615.853} C_VEL
LIN {X 0,Y 450.269,Z 441.112,A -85,B 0,C 180,E1 21612.309,E2 21612.309} C_VEL
LIN {X 0,Y 450.245,Z 441.115,A -85,B 0,C 180,E1 21608.686,E2 21608.686} C_VEL
LIN {X 0,Y 450.227,Z 441.131,A -85,B 0,C 180,E1 21605.097,E2 21605.097} C_VEL
LIN {X 0,Y 450.233,Z 441.149,A -85,B 0,C 180,E1 21601.273,E2 21601.273} C_VEL
LIN {X 0,Y 450.258,Z 441.127,A -85,B 0,C 180,E1 21597.709,E2 21597.709} C_VEL
LIN {X 0,Y 450.291,Z 441.111,A -85,B 0,C 180,E1 21594.009,E2 21594.009} C_VEL
LIN {X 0,Y 450.263,Z 441.113,A -85,B 0,C 180,E1 21590.397,E2 21590.397} C_VEL
LIN {X 0,Y 450.245,Z 441.122,A -85,B 0,C 180,E1 21586.777,E2 21586.777} C_VEL
LIN {X 0,Y 450.254,Z 441.13,A -85,B 0,C 180,E1 21583.087,E2 21583.087} C_VEL
LIN {X 0,Y 450.283,Z 441.135,A -85,B 0,C 180,E1 21579.46,E2 21579.46} C_VEL
LIN {X 0,Y 450.333,Z 441.392,A -85,B 0,C 180,E1 21577.514,E2 21577.514} C_VEL
LIN {X 0,Y 451.809,Z 444.939,A -85,B 0,C 180,E1 21576.248,E2 21576.248} C_VEL
LIN {X 0,Y 453.119,Z 446.823,A -85,B 0,C 180,E1 21575.49,E2 21575.49} C_VEL
LIN {X 0,Y 454.843,Z 450.3,A -85,B 0,C 180,E1 21574.332,E2 21574.332} C_VEL
LIN {X 0,Y 455.777,Z 451.799,A -85,B 0,C 180,E1 21573.802,E2 21573.802} C_VEL
LIN {X 0,Y 457.846,Z 455.706,A -85,B 0,C 180,E1 21572.561,E2 21572.561} C_VEL
LIN {X 0,Y 461.294,Z 462.782,A -85,B 0,C 180,E1 21570.525,E2 21570.525} C_VEL
LIN {X 0,Y 463.176,Z 466.21,A -85,B 0,C 180,E1 21569.623,E2 21569.623} C_VEL
LIN {X 0,Y 473.774,Z 479.706,A -85,B 0,C 180,E1 21567.261,E2 21567.261} C_VEL
LIN {X 0,Y 485.559,Z 495.681,A -85,B 0,C 180,E1 21564.897,E2 21564.897} C_VEL
LIN {X 0,Y 497.085,Z 512.571,A -85,B 0,C 180,E1 21562.774,E2 21562.774} C_VEL
LIN {X 0,Y 508.508,Z 530.464,A -85,B 0,C 180,E1 21560.826,E2 21560.826} C_VEL
LIN {X 0,Y 515.134,Z 541.952,A -85,B 0,C 180,E1 21559.744,E2 21559.744} C_VEL
LIN {X 0,Y 504.932,Z 776.616,A -85,B 0,C 180,E1 21556.096,E2 21556.096} C_VEL
LIN {X 0,Y 501.867,Z 845.237,A -85,B 0,C 180,E1 21555,E2 21555} C_VEL
LIN {X 0,Y 499.7,Z 870.133,A -85,B 0,C 180,E1 21554.43,E2 21554.43} C_VEL
LIN {X 0,Y 497.112,Z 892.995,A -85,B 0,C 180,E1 21553.733,E2 21553.733} C_VEL
LIN {X 0,Y 493.781,Z 916.658,A -85,B 0,C 180,E1 21552.795,E2 21552.795} C_VEL
LIN {X 0,Y 490.499,Z 937.105,A -85,B 0,C 180,E1 21551.805,E2 21551.805} C_VEL
LIN {X 0,Y 486.225,Z 960.218,A -85,B 0,C 180,E1 21550.458,E2 21550.458} C_VEL
LIN {X 0,Y 482.226,Z 980.125,A -85,B 0,C 180,E1 21549.075,E2 21549.075} C_VEL
LIN {X 0,Y 477.532,Z 1001.664,A -85,B 0,C 180,E1 21547.314,E2 21547.314} C_VEL
LIN {X 0,Y 473.505,Z 1019.155,A -85,B 0,C 180,E1 21545.65,E2 21545.65} C_VEL
LIN {X 0,Y 468.645,Z 1039.502,A -85,B 0,C 180,E1 21543.399,E2 21543.399} C_VEL
LIN {X 0,Y 464.778,Z 1055.519,A -85,B 0,C 180,E1 21541.341,E2 21541.341} C_VEL
LIN {X 0,Y 460.714,Z 1072.571,A -85,B 0,C 180,E1 21538.804,E2 21538.804} C_VEL
LIN {X 0,Y 457.584,Z 1086.119,A -85,B 0,C 180,E1 21536.473,E2 21536.473} C_VEL
LIN {X 0,Y 454.475,Z 1100.469,A -85,B 0,C 180,E1 21533.604,E2 21533.604} C_VEL
LIN {X 0,Y 452.373,Z 1111.126,A -85,B 0,C 180,E1 21531.118,E2 21531.118} C_VEL
LIN {X 0,Y 450.491,Z 1122.157,A -85,B 0,C 180,E1 21528.104,E2 21528.104} C_VEL
LIN {X 0,Y 449.314,Z 1130.475,A -85,B 0,C 180,E1 21525.356,E2 21525.356} C_VEL
LIN {X 0,Y 448.516,Z 1137.993,A -85,B 0,C 180,E1 21522.358,E2 21522.358} C_VEL
LIN {X 0,Y 448.116,Z 1143.452,A -85,B 0,C 180,E1 21519.504,E2 21519.504} C_VEL
LIN {X 0,Y 447.979,Z 1147.21,A -85,B 0,C 180,E1 21516.923,E2 21516.923} C_VEL
LIN {X 0,Y 447.937,Z 1150.194,A -85,B 0,C 180,E1 21513.798,E2 21513.798} C_VEL
LIN {X 0,Y 447.939,Z 1151.314,A -85,B 0,C 180,E1 21511.151,E2 21511.151} C_VEL
LIN {X 0,Y 447.94,Z 1151.289,A -85,B 0,C 180,E1 21508.721,E2 21508.721} C_VEL
LIN {X 0,Y 447.938,Z 1149.934,A -85,B 0,C 180,E1 21505.776,E2 21505.776} C_VEL
LIN {X 0,Y 447.983,Z 1147.038,A -85,B 0,C 180,E1 21502.949,E2 21502.949} C_VEL
LIN {X 0,Y 448.132,Z 1143.23,A -85,B 0,C 180,E1 21500.367,E2 21500.367} C_VEL
LIN {X 0,Y 448.597,Z 1137.077,A -85,B 0,C 180,E1 21497.252,E2 21497.252} C_VEL
LIN {X 0,Y 449.377,Z 1129.952,A -85,B 0,C 180,E1 21494.462,E2 21494.462} C_VEL
LIN {X 0,Y 450.701,Z 1120.87,A -85,B 0,C 180,E1 21491.503,E2 21491.503} C_VEL
LIN {X 0,Y 452.562,Z 1110.047,A -85,B 0,C 180,E1 21488.62,E2 21488.62} C_VEL
LIN {X 0,Y 454.992,Z 1098.082,A -85,B 0,C 180,E1 21485.873,E2 21485.873} C_VEL
LIN {X 0,Y 457.899,Z 1084.644,A -85,B 0,C 180,E1 21483.267,E2 21483.267} C_VEL
LIN {X 0,Y 461.293,Z 1070.157,A -85,B 0,C 180,E1 21480.81,E2 21480.81} C_VEL
LIN {X 0,Y 465.123,Z 1053.954,A -85,B 0,C 180,E1 21478.455,E2 21478.455} C_VEL
LIN {X 0,Y 469.158,Z 1037.365,A -85,B 0,C 180,E1 21476.349,E2 21476.349} C_VEL
LIN {X 0,Y 473.697,Z 1018.167,A -85,B 0,C 180,E1 21474.259,E2 21474.259} C_VEL
LIN {X 0,Y 477.828,Z 1000.195,A -85,B 0,C 180,E1 21472.563,E2 21472.563} C_VEL
LIN {X 0,Y 482.537,Z 978.37,A -85,B 0,C 180,E1 21470.804,E2 21470.804} C_VEL
LIN {X 0,Y 486.568,Z 958.277,A -85,B 0,C 180,E1 21469.425,E2 21469.425} C_VEL
LIN {X 0,Y 490.672,Z 935.774,A -85,B 0,C 180,E1 21468.135,E2 21468.135} C_VEL
LIN {X 0,Y 493.967,Z 915.138,A -85,B 0,C 180,E1 21467.146,E2 21467.146} C_VEL
LIN {X 0,Y 497.428,Z 889.919,A -85,B 0,C 180,E1 21466.175,E2 21466.175} C_VEL
LIN {X 0,Y 499.835,Z 868.354,A -85,B 0,C 180,E1 21465.531,E2 21465.531} C_VEL
LIN {X 0,Y 501.996,Z 841.805,A -85,B 0,C 180,E1 21464.947,E2 21464.947} C_VEL
LIN {X 0,Y 511.666,Z 618.238,A -85,B 0,C 180,E1 21461.445,E2 21461.445} C_VEL
LIN {X 0,Y 514.941,Z 541.32,A -85,B 0,C 180,E1 21460.237,E2 21460.237} C_VEL
LIN {X 0,Y 502.732,Z 521.276,A -85,B 0,C 180,E1 21458.229,E2 21458.229} C_VEL
LIN {X 0,Y 490.629,Z 502.972,A -85,B 0,C 180,E1 21456.085,E2 21456.085} C_VEL
LIN {X 0,Y 479.979,Z 488.088,A -85,B 0,C 180,E1 21454.046,E2 21454.046} C_VEL
LIN {X 0,Y 469.808,Z 474.68,A -85,B 0,C 180,E1 21451.93,E2 21451.93} C_VEL
LIN {X 0,Y 462.962,Z 465.852,A -85,B 0,C 180,E1 21450.357,E2 21450.357} C_VEL
LIN {X 0,Y 459.648,Z 459.515,A -85,B 0,C 180,E1 21448.593,E2 21448.593} C_VEL
LIN {X 0,Y 457.746,Z 455.577,A -85,B 0,C 180,E1 21447.446,E2 21447.446} C_VEL
LIN {X 0,Y 455.676,Z 451.487,A -85,B 0,C 180,E1 21446.171,E2 21446.171} C_VEL
LIN {X 0,Y 453.187,Z 447.072,A -85,B 0,C 180,E1 21444.645,E2 21444.645} C_VEL
LIN {X 0,Y 452.163,Z 445.362,A -85,B 0,C 180,E1 21444.01,E2 21444.01} C_VEL
LIN {X 0,Y 450.404,Z 441.865,A -85,B 0,C 180,E1 21442.723,E2 21442.723} C_VEL
LIN {X 0,Y 450.314,Z 441.183,A -85,B 0,C 180,E1 21442.315,E2 21442.315} C_VEL
LIN {X 0,Y 450.279,Z 441.111,A -85,B 0,C 180,E1 21438.515,E2 21438.515} C_VEL
LIN {X 0,Y 450.251,Z 441.119,A -85,B 0,C 180,E1 21434.928,E2 21434.928} C_VEL
LIN {X 0,Y 450.248,Z 441.128,A -85,B 0,C 180,E1 21431.14,E2 21431.14} C_VEL
LIN {X 0,Y 450.267,Z 441.145,A -85,B 0,C 180,E1 21427.529,E2 21427.529} C_VEL
LIN {X 0,Y 450.285,Z 441.13,A -85,B 0,C 180,E1 21423.82,E2 21423.82} C_VEL
LIN {X 0,Y 450.269,Z 441.114,A -85,B 0,C 180,E1 21420.127,E2 21420.127} C_VEL
LIN {X 0,Y 450.232,Z 441.114,A -85,B 0,C 180,E1 21416.562,E2 21416.562} C_VEL
LIN {X 0,Y 450.23,Z 441.124,A -85,B 0,C 180,E1 21412.856,E2 21412.856} C_VEL
LIN {X 0,Y 450.252,Z 441.143,A -85,B 0,C 180,E1 21409.249,E2 21409.249} C_VEL
LIN {X 0,Y 450.28,Z 441.141,A -85,B 0,C 180,E1 21405.509,E2 21405.509} C_VEL
LIN {X 0,Y 450.256,Z 441.132,A -85,B 0,C 180,E1 21401.752,E2 21401.752} C_VEL
LIN {X 0,Y 450.217,Z 441.128,A -85,B 0,C 180,E1 21398.178,E2 21398.178} C_VEL
LIN {X 0,Y 450.269,Z 441.519,A -85,B 0,C 180,E1 21396.459,E2 21396.459} C_VEL
LIN {X 0,Y 452.026,Z 445.247,A -85,B 0,C 180,E1 21395.085,E2 21395.085} C_VEL
LIN {X 0,Y 453.118,Z 447.182,A -85,B 0,C 180,E1 21394.373,E2 21394.373} C_VEL
LIN {X 0,Y 455.544,Z 451.624,A -85,B 0,C 180,E1 21392.835,E2 21392.835} C_VEL
LIN {X 0,Y 458.189,Z 457,A -85,B 0,C 180,E1 21391.165,E2 21391.165} C_VEL
LIN {X 0,Y 460.598,Z 461.75,A -85,B 0,C 180,E1 21389.759,E2 21389.759} C_VEL
LIN {X 0,Y 464.512,Z 469.672,A -85,B 0,C 180,E1 21387.589,E2 21387.589} C_VEL
LIN {X 0,Y 470.104,Z 481.664,A -85,B 0,C 180,E1 21384.652,E2 21384.652} C_VEL
LIN {X 0,Y 472.679,Z 487.361,A -85,B 0,C 180,E1 21383.453,E2 21383.453} C_VEL
LIN {X 0,Y 483.125,Z 502.524,A -85,B 0,C 180,E1 21381.334,E2 21381.334} C_VEL
LIN {X 0,Y 494.693,Z 520.266,A -85,B 0,C 180,E1 21379.185,E2 21379.185} C_VEL
LIN {X 0,Y 505.423,Z 538.328,A -85,B 0,C 180,E1 21377.326,E2 21377.326} C_VEL
LIN {X 0,Y 510.074,Z 546.842,A -85,B 0,C 180,E1 21376.552,E2 21376.552} C_VEL
LIN {X 0,Y 512.463,Z 562.501,A -85,B 0,C 180,E1 21375.939,E2 21375.939} C_VEL
LIN {X 0,Y 502.677,Z 820.303,A -85,B 0,C 180,E1 21372.149,E2 21372.149} C_VEL
LIN {X 0,Y 501.129,Z 852.998,A -85,B 0,C 180,E1 21371.624,E2 21371.624} C_VEL
LIN {X 0,Y 499.186,Z 874.931,A -85,B 0,C 180,E1 21371.112,E2 21371.112} C_VEL
LIN {X 0,Y 496.327,Z 899.32,A -85,B 0,C 180,E1 21370.33,E2 21370.33} C_VEL
LIN {X 0,Y 493.335,Z 919.859,A -85,B 0,C 180,E1 21369.484,E2 21369.484} C_VEL
LIN {X 0,Y 489.613,Z 941.531,A -85,B 0,C 180,E1 21368.377,E2 21368.377} C_VEL
LIN {X 0,Y 485.904,Z 960.471,A -85,B 0,C 180,E1 21367.215,E2 21367.215} C_VEL
LIN {X 0,Y 481.442,Z 981.085,A -85,B 0,C 180,E1 21365.702,E2 21365.702} C_VEL
LIN {X 0,Y 477.213,Z 999.109,A -85,B 0,C 180,E1 21364.143,E2 21364.143} C_VEL
LIN {X 0,Y 472.636,Z 1017.322,A -85,B 0,C 180,E1 21362.288,E2 21362.288} C_VEL
LIN {X 0,Y 468.492,Z 1033.364,A -85,B 0,C 180,E1 21360.386,E2 21360.386} C_VEL
LIN {X 0,Y 464.196,Z 1049.455,A -85,B 0,C 180,E1 21358.147,E2 21358.147} C_VEL
LIN {X 0,Y 460.499,Z 1063.514,A -85,B 0,C 180,E1 21355.877,E2 21355.877} C_VEL
LIN {X 0,Y 457.035,Z 1076.838,A -85,B 0,C 180,E1 21353.328,E2 21353.328} C_VEL
LIN {X 0,Y 454.14,Z 1088.883,A -85,B 0,C 180,E1 21350.627,E2 21350.627} C_VEL
LIN {X 0,Y 451.893,Z 1098.917,A -85,B 0,C 180,E1 21347.912,E2 21347.912} C_VEL
LIN {X 0,Y 451.739,Z 1099.709,A -85,B 0,C 180,E1 21347.682,E2 21347.682} C_VEL
LIN {X 0,Y 450.191,Z 1102.796,A -85,B 0,C 180,E1 21346.797,E2 21346.797} C_VEL
LIN {X 0,Y 442.705,Z 1110.335,A -85,B 0,C 180,E1 21344.432,E2 21344.432} C_VEL
LIN {X 0,Y 441.6,Z 1112.327,A -85,B 0,C 180,E1 21343.619,E2 21343.619} C_VEL
LIN {X 0,Y 440.704,Z 1118.366,A -85,B 0,C 180,E1 21340.722,E2 21340.722} C_VEL
LIN {X 0,Y 440.226,Z 1123.168,A -85,B 0,C 180,E1 21337.701,E2 21337.701} C_VEL
LIN {X 0,Y 440.014,Z 1126.17,A -85,B 0,C 180,E1 21334.823,E2 21334.823} C_VEL
LIN {X 0,Y 439.953,Z 1127.927,A -85,B 0,C 180,E1 21331.823,E2 21331.823} C_VEL
LIN {X 0,Y 439.951,Z 1128.094,A -85,B 0,C 180,E1 21329.088,E2 21329.088} C_VEL
LIN {X 0,Y 439.978,Z 1127.104,A -85,B 0,C 180,E1 21326.352,E2 21326.352} C_VEL
LIN {X 0,Y 440.126,Z 1124.357,A -85,B 0,C 180,E1 21323.215,E2 21323.215} C_VEL
LIN {X 0,Y 440.456,Z 1120.602,A -85,B 0,C 180,E1 21320.461,E2 21320.461} C_VEL
LIN {X 0,Y 441.235,Z 1114.591,A -85,B 0,C 180,E1 21317.302,E2 21317.302} C_VEL
LIN {X 0,Y 442.456,Z 1107.503,A -85,B 0,C 180,E1 21314.4,E2 21314.4} C_VEL
LIN {X 0,Y 444.272,Z 1098.583,A -85,B 0,C 180,E1 21311.498,E2 21311.498} C_VEL
LIN {X 0,Y 446.689,Z 1088.474,A -85,B 0,C 180,E1 21308.738,E2 21308.738} C_VEL
LIN {X 0,Y 449.732,Z 1076.479,A -85,B 0,C 180,E1 21306.033,E2 21306.033} C_VEL
LIN {X 0,Y 453.446,Z 1062.815,A -85,B 0,C 180,E1 21303.408,E2 21303.408} C_VEL
LIN {X 0,Y 457.132,Z 1049.492,A -85,B 0,C 180,E1 21301.235,E2 21301.235} C_VEL
LIN {X 0,Y 461.687,Z 1033.058,A -85,B 0,C 180,E1 21298.927,E2 21298.927} C_VEL
LIN {X 0,Y 465.924,Z 1017.341,A -85,B 0,C 180,E1 21297.046,E2 21297.046} C_VEL
LIN {X 0,Y 471.054,Z 997.584,A -85,B 0,C 180,E1 21295.032,E2 21295.032} C_VEL
LIN {X 0,Y 475.256,Z 980.28,A -85,B 0,C 180,E1 21293.533,E2 21293.533} C_VEL
LIN {X 0,Y 479.912,Z 959.31,A -85,B 0,C 180,E1 21291.999,E2 21291.999} C_VEL
LIN {X 0,Y 483.88,Z 939.63,A -85,B 0,C 180,E1 21290.796,E2 21290.796} C_VEL
LIN {X 0,Y 487.756,Z 917.237,A -85,B 0,C 180,E1 21289.675,E2 21289.675} C_VEL
LIN {X 0,Y 491.011,Z 895.382,A -85,B 0,C 180,E1 21288.793,E2 21288.793} C_VEL
LIN {X 0,Y 493.644,Z 872.531,A -85,B 0,C 180,E1 21288.093,E2 21288.093} C_VEL
LIN {X 0,Y 495.692,Z 849.194,A -85,B 0,C 180,E1 21287.566,E2 21287.566} C_VEL
LIN {X 0,Y 498.236,Z 787.558,A -85,B 0,C 180,E1 21286.628,E2 21286.628} C_VEL
LIN {X 0,Y 507.095,Z 562.905,A -85,B 0,C 180,E1 21283.286,E2 21283.286} C_VEL
LIN {X 0,Y 504.917,Z 550.379,A -85,B 0,C 180,E1 21282.746,E2 21282.746} C_VEL
LIN {X 0,Y 493.383,Z 530.358,A -85,B 0,C 180,E1 21280.736,E2 21280.736} C_VEL
LIN {X 0,Y 481.876,Z 512.107,A -85,B 0,C 180,E1 21278.575,E2 21278.575} C_VEL
LIN {X 0,Y 472.528,Z 498.289,A -85,B 0,C 180,E1 21276.677,E2 21276.677} C_VEL
LIN {X 0,Y 463.769,Z 485.674,A -85,B 0,C 180,E1 21274.694,E2 21274.694} C_VEL
LIN {X 0,Y 458.565,Z 474.269,A -85,B 0,C 180,E1 21271.849,E2 21271.849} C_VEL
LIN {X 0,Y 454.151,Z 465.403,A -85,B 0,C 180,E1 21269.324,E2 21269.324} C_VEL
LIN {X 0,Y 451.724,Z 460.631,A -85,B 0,C 180,E1 21267.843,E2 21267.843} C_VEL
LIN {X 0,Y 449.541,Z 456.26,A -85,B 0,C 180,E1 21266.414,E2 21266.414} C_VEL
LIN {X 0,Y 447.048,Z 451.514,A -85,B 0,C 180,E1 21264.725,E2 21264.725} C_VEL
LIN {X 0,Y 445.052,Z 447.547,A -85,B 0,C 180,E1 21263.234,E2 21263.234} C_VEL
LIN {X 0,Y 442.483,Z 443.206,A -85,B 0,C 180,E1 21261.335,E2 21261.335} C_VEL
LIN {X 0,Y 442.312,Z 442.184,A -85,B 0,C 180,E1 21260.788,E2 21260.788} C_VEL
LIN {X 0,Y 442.28,Z 442.108,A -85,B 0,C 180,E1 21257.092,E2 21257.092} C_VEL
LIN {X 0,Y 442.276,Z 442.114,A -85,B 0,C 180,E1 21253.466,E2 21253.466} C_VEL
LIN {X 0,Y 442.295,Z 442.124,A -85,B 0,C 180,E1 21249.762,E2 21249.762} C_VEL
LIN {X 0,Y 442.335,Z 442.13,A -85,B 0,C 180,E1 21246.099,E2 21246.099} C_VEL
LIN {X 0,Y 442.334,Z 442.111,A -85,B 0,C 180,E1 21242.332,E2 21242.332} C_VEL
LIN {X 0,Y 442.298,Z 442.102,A -85,B 0,C 180,E1 21238.834,E2 21238.834} C_VEL
LIN {X 0,Y 442.296,Z 442.106,A -85,B 0,C 180,E1 21235.202,E2 21235.202} C_VEL
LIN {X 0,Y 442.324,Z 442.117,A -85,B 0,C 180,E1 21231.551,E2 21231.551} C_VEL
LIN {X 0,Y 442.354,Z 442.13,A -85,B 0,C 180,E1 21227.865,E2 21227.865} C_VEL
LIN {X 0,Y 442.336,Z 442.119,A -85,B 0,C 180,E1 21224.261,E2 21224.261} C_VEL
LIN {X 0,Y 442.319,Z 442.112,A -85,B 0,C 180,E1 21220.591,E2 21220.591} C_VEL
LIN {X 0,Y 442.432,Z 442.595,A -85,B 0,C 180,E1 21219.733,E2 21219.733} C_VEL
LIN {X 0,Y 443.997,Z 446.08,A -85,B 0,C 180,E1 21218.325,E2 21218.325} C_VEL
LIN {X 0,Y 445.227,Z 447.744,A -85,B 0,C 180,E1 21217.556,E2 21217.556} C_VEL
LIN {X 0,Y 446.947,Z 451.322,A -85,B 0,C 180,E1 21216.254,E2 21216.254} C_VEL
LIN {X 0,Y 448.012,Z 453.045,A -85,B 0,C 180,E1 21215.588,E2 21215.588} C_VEL
LIN {X 0,Y 449.963,Z 456.68,A -85,B 0,C 180,E1 21214.321,E2 21214.321} C_VEL
LIN {X 0,Y 453.253,Z 463.202,A -85,B 0,C 180,E1 21212.259,E2 21212.259} C_VEL
LIN {X 0,Y 455.394,Z 466.921,A -85,B 0,C 180,E1 21211.187,E2 21211.187} C_VEL
LIN {X 0,Y 465.546,Z 479.845,A -85,B 0,C 180,E1 21208.755,E2 21208.755} C_VEL
LIN {X 0,Y 475.524,Z 493.031,A -85,B 0,C 180,E1 21206.606,E2 21206.606} C_VEL
LIN {X 0,Y 486.38,Z 508.308,A -85,B 0,C 180,E1 21204.46,E2 21204.46} C_VEL
LIN {X 0,Y 498.319,Z 526.415,A -85,B 0,C 180,E1 21202.284,E2 21202.284} C_VEL
LIN {X 0,Y 509.645,Z 545.145,A -85,B 0,C 180,E1 21200.364,E2 21200.364} C_VEL
LIN {X 0,Y 499.153,Z 778.594,A -85,B 0,C 180,E1 21196.709,E2 21196.709} C_VEL
LIN {X 0,Y 496.059,Z 845.371,A -85,B 0,C 180,E1 21195.633,E2 21195.633} C_VEL
LIN {X 0,Y 493.833,Z 870.215,A -85,B 0,C 180,E1 21195.06,E2 21195.06} C_VEL
LIN {X 0,Y 491.196,Z 892.845,A -85,B 0,C 180,E1 21194.366,E2 21194.366} C_VEL
LIN {X 0,Y 487.838,Z 916.056,A -85,B 0,C 180,E1 21193.445,E2 21193.445} C_VEL
LIN {X 0,Y 484.442,Z 936.568,A -85,B 0,C 180,E1 21192.449,E2 21192.449} C_VEL
LIN {X 0,Y 480.004,Z 959.842,A -85,B 0,C 180,E1 21191.088,E2 21191.088} C_VEL
LIN {X 0,Y 476.029,Z 978.961,A -85,B 0,C 180,E1 21189.755,E2 21189.755} C_VEL
LIN {X 0,Y 471.025,Z 1001.18,A -85,B 0,C 180,E1 21187.934,E2 21187.934} C_VEL
LIN {X 0,Y 466.808,Z 1018.816,A -85,B 0,C 180,E1 21186.241,E2 21186.241} C_VEL
LIN {X 0,Y 461.76,Z 1039.167,A -85,B 0,C 180,E1 21183.968,E2 21183.968} C_VEL
LIN {X 0,Y 457.759,Z 1055.009,A -85,B 0,C 180,E1 21181.911,E2 21181.911} C_VEL
LIN {X 0,Y 453.453,Z 1072.296,A -85,B 0,C 180,E1 21179.309,E2 21179.309} C_VEL
LIN {X 0,Y 450.163,Z 1085.853,A -85,B 0,C 180,E1 21176.944,E2 21176.944} C_VEL
LIN {X 0,Y 446.891,Z 1100.217,A -85,B 0,C 180,E1 21174.03,E2 21174.03} C_VEL
LIN {X 0,Y 444.661,Z 1110.88,A -85,B 0,C 180,E1 21171.502,E2 21171.502} C_VEL
LIN {X 0,Y 442.666,Z 1121.93,A -85,B 0,C 180,E1 21168.432,E2 21168.432} C_VEL
LIN {X 0,Y 441.416,Z 1130.245,A -85,B 0,C 180,E1 21165.638,E2 21165.638} C_VEL
LIN {X 0,Y 440.563,Z 1137.771,A -85,B 0,C 180,E1 21162.585,E2 21162.585} C_VEL
LIN {X 0,Y 440.128,Z 1143.349,A -85,B 0,C 180,E1 21159.607,E2 21159.607} C_VEL
LIN {X 0,Y 439.978,Z 1147.161,A -85,B 0,C 180,E1 21156.918,E2 21156.918} C_VEL
LIN {X 0,Y 439.939,Z 1150.031,A -85,B 0,C 180,E1 21153.779,E2 21153.779} C_VEL
LIN {X 0,Y 439.941,Z 1151.104,A -85,B 0,C 180,E1 21151.172,E2 21151.172} C_VEL
LIN {X 0,Y 439.943,Z 1151.079,A -85,B 0,C 180,E1 21148.698,E2 21148.698} C_VEL
LIN {X 0,Y 439.94,Z 1149.721,A -85,B 0,C 180,E1 21145.699,E2 21145.699} C_VEL
LIN {X 0,Y 439.98,Z 1146.822,A -85,B 0,C 180,E1 21142.82,E2 21142.82} C_VEL
LIN {X 0,Y 440.149,Z 1143.011,A -85,B 0,C 180,E1 21140.19,E2 21140.19} C_VEL
LIN {X 0,Y 440.647,Z 1136.851,A -85,B 0,C 180,E1 21137.018,E2 21137.018} C_VEL
LIN {X 0,Y 441.464,Z 1129.862,A -85,B 0,C 180,E1 21134.229,E2 21134.229} C_VEL
LIN {X 0,Y 442.816,Z 1121.067,A -85,B 0,C 180,E1 21131.298,E2 21131.298} C_VEL
LIN {X 0,Y 444.759,Z 1110.328,A -85,B 0,C 180,E1 21128.365,E2 21128.365} C_VEL
LIN {X 0,Y 447.157,Z 1099.01,A -85,B 0,C 180,E1 21125.704,E2 21125.704} C_VEL
LIN {X 0,Y 450.332,Z 1085.065,A -85,B 0,C 180,E1 21122.919,E2 21122.919} C_VEL
LIN {X 0,Y 453.714,Z 1071.199,A -85,B 0,C 180,E1 21120.517,E2 21120.517} C_VEL
LIN {X 0,Y 457.867,Z 1054.47,A -85,B 0,C 180,E1 21118.023,E2 21118.023} C_VEL
LIN {X 0,Y 461.878,Z 1038.603,A -85,B 0,C 180,E1 21115.971,E2 21115.971} C_VEL
LIN {X 0,Y 466.794,Z 1018.716,A -85,B 0,C 180,E1 21113.757,E2 21113.757} C_VEL
LIN {X 0,Y 471.14,Z 1000.508,A -85,B 0,C 180,E1 21112.014,E2 21112.014} C_VEL
LIN {X 0,Y 475.991,Z 978.911,A -85,B 0,C 180,E1 21110.25,E2 21110.25} C_VEL
LIN {X 0,Y 479.987,Z 959.683,A -85,B 0,C 180,E1 21108.91,E2 21108.91} C_VEL
LIN {X 0,Y 484.424,Z 936.364,A -85,B 0,C 180,E1 21107.549,E2 21107.549} C_VEL
LIN {X 0,Y 487.819,Z 915.814,A -85,B 0,C 180,E1 21106.553,E2 21106.553} C_VEL
LIN {X 0,Y 491.411,Z 890.623,A -85,B 0,C 180,E1 21105.569,E2 21105.569} C_VEL
LIN {X 0,Y 493.9,Z 869.053,A -85,B 0,C 180,E1 21104.918,E2 21104.918} C_VEL
LIN {X 0,Y 496.133,Z 842.903,A -85,B 0,C 180,E1 21104.331,E2 21104.331} C_VEL
LIN {X 0,Y 505.69,Z 629.764,A -85,B 0,C 180,E1 21100.965,E2 21100.965} C_VEL
LIN {X 0,Y 509.411,Z 544.834,A -85,B 0,C 180,E1 21099.619,E2 21099.619} C_VEL
LIN {X 0,Y 497.603,Z 525.382,A -85,B 0,C 180,E1 21097.616,E2 21097.616} C_VEL
LIN {X 0,Y 485.419,Z 506.916,A -85,B 0,C 180,E1 21095.386,E2 21095.386} C_VEL
LIN {X 0,Y 473.516,Z 490.294,A -85,B 0,C 180,E1 21093.011,E2 21093.011} C_VEL
LIN {X 0,Y 463.026,Z 476.633,A -85,B 0,C 180,E1 21090.712,E2 21090.712} C_VEL
LIN {X 0,Y 457.762,Z 470.196,A -85,B 0,C 180,E1 21089.473,E2 21089.473} C_VEL
LIN {X 0,Y 455.072,Z 466.387,A -85,B 0,C 180,E1 21088.754,E2 21088.754} C_VEL
LIN {X 0,Y 452.088,Z 460.99,A -85,B 0,C 180,E1 21087.105,E2 21087.105} C_VEL
LIN {X 0,Y 449.858,Z 456.544,A -85,B 0,C 180,E1 21085.685,E2 21085.685} C_VEL
LIN {X 0,Y 447.906,Z 452.718,A -85,B 0,C 180,E1 21084.382,E2 21084.382} C_VEL
LIN {X 0,Y 445.353,Z 448.214,A -85,B 0,C 180,E1 21082.666,E2 21082.666} C_VEL
LIN {X 0,Y 444.538,Z 446.672,A -85,B 0,C 180,E1 21082.063,E2 21082.063} C_VEL
LIN {X 0,Y 442.592,Z 443.353,A -85,B 0,C 180,E1 21080.636,E2 21080.636} C_VEL
LIN {X 0,Y 442.369,Z 442.193,A -85,B 0,C 180,E1 21080.094,E2 21080.094} C_VEL
LIN {X 0,Y 442.356,Z 442.129,A -85,B 0,C 180,E1 21076.277,E2 21076.277} C_VEL
LIN {X 0,Y 442.319,Z 442.12,A -85,B 0,C 180,E1 21072.666,E2 21072.666} C_VEL
LIN {X 0,Y 442.307,Z 442.109,A -85,B 0,C 180,E1 21068.923,E2 21068.923} C_VEL
LIN {X 0,Y 442.306,Z 442.102,A -85,B 0,C 180,E1 21065.188,E2 21065.188} C_VEL
LIN {X 0,Y 442.329,Z 442.102,A -85,B 0,C 180,E1 21061.554,E2 21061.554} C_VEL
LIN {X 0,Y 442.34,Z 442.118,A -85,B 0,C 180,E1 21057.927,E2 21057.927} C_VEL
LIN {X 0,Y 442.316,Z 442.133,A -85,B 0,C 180,E1 21054.161,E2 21054.161} C_VEL
LIN {X 0,Y 442.288,Z 442.117,A -85,B 0,C 180,E1 21050.501,E2 21050.501} C_VEL
LIN {X 0,Y 442.284,Z 442.109,A -85,B 0,C 180,E1 21046.801,E2 21046.801} C_VEL
LIN {X 0,Y 442.318,Z 442.103,A -85,B 0,C 180,E1 21043.316,E2 21043.316} C_VEL
LIN {X 0,Y 442.324,Z 442.105,A -85,B 0,C 180,E1 21039.627,E2 21039.627} C_VEL
LIN {X 0,Y 442.345,Z 442.559,A -85,B 0,C 180,E1 21038.728,E2 21038.728} C_VEL
LIN {X 0,Y 444.072,Z 446.222,A -85,B 0,C 180,E1 21037.214,E2 21037.214} C_VEL
LIN {X 0,Y 445.201,Z 448.044,A -85,B 0,C 180,E1 21036.436,E2 21036.436} C_VEL
LIN {X 0,Y 447.944,Z 453.291,A -85,B 0,C 180,E1 21034.481,E2 21034.481} C_VEL
LIN {X 0,Y 450.33,Z 457.784,A -85,B 0,C 180,E1 21032.919,E2 21032.919} C_VEL
LIN {X 0,Y 452.772,Z 462.668,A -85,B 0,C 180,E1 21031.366,E2 21031.366} C_VEL
LIN {X 0,Y 455.338,Z 467.91,A -85,B 0,C 180,E1 21029.81,E2 21029.81} C_VEL
LIN {X 0,Y 458.998,Z 475.358,A -85,B 0,C 180,E1 21027.743,E2 21027.743} C_VEL
LIN {X 0,Y 464.172,Z 486.371,A -85,B 0,C 180,E1 21025.04,E2 21025.04} C_VEL
LIN {X 0,Y 477.567,Z 505.626,A -85,B 0,C 180,E1 21022.16,E2 21022.16} C_VEL
LIN {X 0,Y 488.279,Z 522.28,A -85,B 0,C 180,E1 21020.079,E2 21020.079} C_VEL
LIN {X 0,Y 498.395,Z 538.994,A -85,B 0,C 180,E1 21018.257,E2 21018.257} C_VEL
LIN {X 0,Y 505.12,Z 551.106,A -85,B 0,C 180,E1 21017.101,E2 21017.101} C_VEL
LIN {X 0,Y 507.044,Z 564.058,A -85,B 0,C 180,E1 21016.587,E2 21016.587} C_VEL
LIN {X 0,Y 496.876,Z 821.748,A -85,B 0,C 180,E1 21012.768,E2 21012.768} C_VEL
LIN {X 0,Y 495.279,Z 853.591,A -85,B 0,C 180,E1 21012.248,E2 21012.248} C_VEL
LIN {X 0,Y 493.274,Z 875.444,A -85,B 0,C 180,E1 21011.732,E2 21011.732} C_VEL
LIN {X 0,Y 490.381,Z 899.282,A -85,B 0,C 180,E1 21010.961,E2 21010.961} C_VEL
LIN {X 0,Y 487.303,Z 919.767,A -85,B 0,C 180,E1 21010.113,E2 21010.113} C_VEL
LIN {X 0,Y 483.356,Z 942.017,A -85,B 0,C 180,E1 21008.967,E2 21008.967} C_VEL
LIN {X 0,Y 479.491,Z 961.111,A -85,B 0,C 180,E1 21007.783,E2 21007.783} C_VEL
LIN {X 0,Y 474.852,Z 981.75,A -85,B 0,C 180,E1 21006.246,E2 21006.246} C_VEL
LIN {X 0,Y 470.463,Z 999.813,A -85,B 0,C 180,E1 21004.663,E2 21004.663} C_VEL
LIN {X 0,Y 465.655,Z 1018.185,A -85,B 0,C 180,E1 21002.76,E2 21002.76} C_VEL
LIN {X 0,Y 461.125,Z 1035.109,A -85,B 0,C 180,E1 21000.714,E2 21000.714} C_VEL
LIN {X 0,Y 456.801,Z 1050.56,A -85,B 0,C 180,E1 20998.502,E2 20998.502} C_VEL
LIN {X 0,Y 452.782,Z 1065.206,A -85,B 0,C 180,E1 20996.069,E2 20996.069} C_VEL
LIN {X 0,Y 449.39,Z 1077.71,A -85,B 0,C 180,E1 20993.61,E2 20993.61} C_VEL
LIN {X 0,Y 446.382,Z 1089.624,A -85,B 0,C 180,E1 20990.865,E2 20990.865} C_VEL
LIN {X 0,Y 444.094,Z 1099.384,A -85,B 0,C 180,E1 20988.167,E2 20988.167} C_VEL
LIN {X 0,Y 442.235,Z 1108.617,A -85,B 0,C 180,E1 20985.071,E2 20985.071} C_VEL
LIN {X 0,Y 441.6,Z 1112.327,A -85,B 0,C 180,E1 20983.619,E2 20983.619} C_VEL
LIN {X 0,Y 440.248,Z 1114.542,A -85,B 0,C 180,E1 20982.666,E2 20982.666} C_VEL
LIN {X 0,Y 433.211,Z 1120.124,A -85,B 0,C 180,E1 20980.054,E2 20980.054} C_VEL
LIN {X 0,Y 432.439,Z 1121.337,A -85,B 0,C 180,E1 20979.268,E2 20979.268} C_VEL
LIN {X 0,Y 432.112,Z 1125.071,A -85,B 0,C 180,E1 20976.377,E2 20976.377} C_VEL
LIN {X 0,Y 431.975,Z 1127.46,A -85,B 0,C 180,E1 20973.317,E2 20973.317} C_VEL
LIN {X 0,Y 431.954,Z 1128.331,A -85,B 0,C 180,E1 20970.663,E2 20970.663} C_VEL
LIN {X 0,Y 431.961,Z 1127.901,A -85,B 0,C 180,E1 20967.479,E2 20967.479} C_VEL
LIN {X 0,Y 432.04,Z 1126.136,A -85,B 0,C 180,E1 20964.688,E2 20964.688} C_VEL
LIN {X 0,Y 432.295,Z 1122.807,A -85,B 0,C 180,E1 20961.621,E2 20961.621} C_VEL
LIN {X 0,Y 432.851,Z 1118.029,A -85,B 0,C 180,E1 20958.676,E2 20958.676} C_VEL
LIN {X 0,Y 433.914,Z 1111.487,A -85,B 0,C 180,E1 20955.589,E2 20955.589} C_VEL
LIN {X 0,Y 435.419,Z 1103.867,A -85,B 0,C 180,E1 20952.768,E2 20952.768} C_VEL
LIN {X 0,Y 437.785,Z 1093.722,A -85,B 0,C 180,E1 20949.686,E2 20949.686} C_VEL
LIN {X 0,Y 440.536,Z 1083.141,A -85,B 0,C 180,E1 20947.021,E2 20947.021} C_VEL
LIN {X 0,Y 444.226,Z 1069.825,A -85,B 0,C 180,E1 20944.204,E2 20944.204} C_VEL
LIN {X 0,Y 448.132,Z 1056.294,A -85,B 0,C 180,E1 20941.769,E2 20941.769} C_VEL
LIN {X 0,Y 452.509,Z 1041.081,A -85,B 0,C 180,E1 20939.454,E2 20939.454} C_VEL
LIN {X 0,Y 457.232,Z 1024.699,A -85,B 0,C 180,E1 20937.306,E2 20937.306} C_VEL
LIN {X 0,Y 461.971,Z 1007.25,A -85,B 0,C 180,E1 20935.378,E2 20935.378} C_VEL
LIN {X 0,Y 466.853,Z 988.624,A -85,B 0,C 180,E1 20933.61,E2 20933.61} C_VEL
LIN {X 0,Y 471.355,Z 969.724,A -85,B 0,C 180,E1 20932.104,E2 20932.104} C_VEL
LIN {X 0,Y 475.965,Z 948.832,A -85,B 0,C 180,E1 20930.7,E2 20930.7} C_VEL
LIN {X 0,Y 479.781,Z 928.976,A -85,B 0,C 180,E1 20929.598,E2 20929.598} C_VEL
LIN {X 0,Y 483.397,Z 907.51,A -85,B 0,C 180,E1 20928.614,E2 20928.614} C_VEL
LIN {X 0,Y 486.308,Z 886.215,A -85,B 0,C 180,E1 20927.846,E2 20927.846} C_VEL
LIN {X 0,Y 488.822,Z 863.287,A -85,B 0,C 180,E1 20927.211,E2 20927.211} C_VEL
LIN {X 0,Y 490.434,Z 840.754,A -85,B 0,C 180,E1 20926.772,E2 20926.772} C_VEL
LIN {X 0,Y 500.609,Z 592.271,A -85,B 0,C 180,E1 20923.049,E2 20923.049} C_VEL
LIN {X 0,Y 501.691,Z 564.252,A -85,B 0,C 180,E1 20922.611,E2 20922.611} C_VEL
LIN {X 0,Y 500.048,Z 554.763,A -85,B 0,C 180,E1 20922.192,E2 20922.192} C_VEL
LIN {X 0,Y 489.143,Z 535.721,A -85,B 0,C 180,E1 20920.238,E2 20920.238} C_VEL
LIN {X 0,Y 478.182,Z 518.155,A -85,B 0,C 180,E1 20918.125,E2 20918.125} C_VEL
LIN {X 0,Y 469.197,Z 504.686,A -85,B 0,C 180,E1 20916.255,E2 20916.255} C_VEL
LIN {X 0,Y 459.541,Z 491.058,A -85,B 0,C 180,E1 20914.075,E2 20914.075} C_VEL
LIN {X 0,Y 455.395,Z 484.924,A -85,B 0,C 180,E1 20912.992,E2 20912.992} C_VEL
LIN {X 0,Y 450.323,Z 474.456,A -85,B 0,C 180,E1 20910.12,E2 20910.12} C_VEL
LIN {X 0,Y 448.375,Z 470.526,A -85,B 0,C 180,E1 20908.942,E2 20908.942} C_VEL
LIN {X 0,Y 446.314,Z 466.341,A -85,B 0,C 180,E1 20907.629,E2 20907.629} C_VEL
LIN {X 0,Y 444.146,Z 462.009,A -85,B 0,C 180,E1 20906.184,E2 20906.184} C_VEL
LIN {X 0,Y 441.744,Z 457.359,A -85,B 0,C 180,E1 20904.504,E2 20904.504} C_VEL
LIN {X 0,Y 439.436,Z 452.881,A -85,B 0,C 180,E1 20902.757,E2 20902.757} C_VEL
LIN {X 0,Y 437.364,Z 449.15,A -85,B 0,C 180,E1 20901.13,E2 20901.13} C_VEL
LIN {X 0,Y 436.45,Z 447.545,A -85,B 0,C 180,E1 20900.379,E2 20900.379} C_VEL
LIN {X 0,Y 434.624,Z 444.377,A -85,B 0,C 180,E1 20898.789,E2 20898.789} C_VEL
LIN {X 0,Y 434.378,Z 443.219,A -85,B 0,C 180,E1 20898.105,E2 20898.105} C_VEL
LIN {X 0,Y 434.404,Z 443.115,A -85,B 0,C 180,E1 20894.394,E2 20894.394} C_VEL
LIN {X 0,Y 434.389,Z 443.121,A -85,B 0,C 180,E1 20890.477,E2 20890.477} C_VEL
LIN {X 0,Y 434.356,Z 443.103,A -85,B 0,C 180,E1 20886.875,E2 20886.875} C_VEL
LIN {X 0,Y 434.348,Z 443.092,A -85,B 0,C 180,E1 20883.167,E2 20883.167} C_VEL
LIN {X 0,Y 434.36,Z 443.09,A -85,B 0,C 180,E1 20879.472,E2 20879.472} C_VEL
LIN {X 0,Y 434.389,Z 443.099,A -85,B 0,C 180,E1 20875.776,E2 20875.776} C_VEL
LIN {X 0,Y 434.422,Z 443.114,A -85,B 0,C 180,E1 20872.062,E2 20872.062} C_VEL
LIN {X 0,Y 434.405,Z 443.117,A -85,B 0,C 180,E1 20868.179,E2 20868.179} C_VEL
LIN {X 0,Y 434.38,Z 443.103,A -85,B 0,C 180,E1 20864.513,E2 20864.513} C_VEL
LIN {X 0,Y 434.442,Z 443.482,A -85,B 0,C 180,E1 20862.465,E2 20862.465} C_VEL
LIN {X 0,Y 436.322,Z 447.407,A -85,B 0,C 180,E1 20860.592,E2 20860.592} C_VEL
LIN {X 0,Y 437.414,Z 448.92,A -85,B 0,C 180,E1 20859.808,E2 20859.808} C_VEL
LIN {X 0,Y 439.144,Z 452.444,A -85,B 0,C 180,E1 20858.355,E2 20858.355} C_VEL
LIN {X 0,Y 440.145,Z 453.856,A -85,B 0,C 180,E1 20857.705,E2 20857.705} C_VEL
LIN {X 0,Y 442.083,Z 457.7,A -85,B 0,C 180,E1 20856.259,E2 20856.259} C_VEL
LIN {X 0,Y 443.164,Z 459.945,A -85,B 0,C 180,E1 20855.471,E2 20855.471} C_VEL
LIN {X 0,Y 445.401,Z 464.002,A -85,B 0,C 180,E1 20854.039,E2 20854.039} C_VEL
LIN {X 0,Y 447.379,Z 467.539,A -85,B 0,C 180,E1 20852.946,E2 20852.946} C_VEL
LIN {X 0,Y 453.41,Z 475.075,A -85,B 0,C 180,E1 20851.338,E2 20851.338} C_VEL
LIN {X 0,Y 458.179,Z 481.086,A -85,B 0,C 180,E1 20850.161,E2 20850.161} C_VEL
LIN {X 0,Y 466.241,Z 491.355,A -85,B 0,C 180,E1 20848.303,E2 20848.303} C_VEL
LIN {X 0,Y 476.407,Z 505.439,A -85,B 0,C 180,E1 20846.135,E2 20846.135} C_VEL
LIN {X 0,Y 486.545,Z 520.154,A -85,B 0,C 180,E1 20844.147,E2 20844.147} C_VEL
LIN {X 0,Y 499.192,Z 540.198,A -85,B 0,C 180,E1 20841.853,E2 20841.853} C_VEL
LIN {X 0,Y 504.187,Z 549.057,A -85,B 0,C 180,E1 20840.986,E2 20840.986} C_VEL
LIN {X 0,Y 493.327,Z 782.8,A -85,B 0,C 180,E1 20837.3,E2 20837.3} C_VEL
LIN {X 0,Y 490.303,Z 845.693,A -85,B 0,C 180,E1 20836.278,E2 20836.278} C_VEL
LIN {X 0,Y 488.021,Z 870.363,A -85,B 0,C 180,E1 20835.703,E2 20835.703} C_VEL
LIN {X 0,Y 485.299,Z 893.043,A -85,B 0,C 180,E1 20835.003,E2 20835.003} C_VEL
LIN {X 0,Y 481.744,Z 916.751,A -85,B 0,C 180,E1 20834.053,E2 20834.053} C_VEL
LIN {X 0,Y 478.045,Z 938.314,A -85,B 0,C 180,E1 20832.99,E2 20832.99} C_VEL
LIN {X 0,Y 473.667,Z 960.312,A -85,B 0,C 180,E1 20831.679,E2 20831.679} C_VEL
LIN {X 0,Y 469.396,Z 980.129,A -85,B 0,C 180,E1 20830.279,E2 20830.279} C_VEL
LIN {X 0,Y 464.348,Z 1001.628,A -85,B 0,C 180,E1 20828.485,E2 20828.485} C_VEL
LIN {X 0,Y 459.861,Z 1019.717,A -85,B 0,C 180,E1 20826.723,E2 20826.723} C_VEL
LIN {X 0,Y 454.908,Z 1038.891,A -85,B 0,C 180,E1 20824.547,E2 20824.547} C_VEL
LIN {X 0,Y 450.738,Z 1054.717,A -85,B 0,C 180,E1 20822.469,E2 20822.469} C_VEL
LIN {X 0,Y 446.227,Z 1072.024,A -85,B 0,C 180,E1 20819.832,E2 20819.832} C_VEL
LIN {X 0,Y 442.776,Z 1085.588,A -85,B 0,C 180,E1 20817.431,E2 20817.431} C_VEL
LIN {X 0,Y 439.285,Z 1100.15,A -85,B 0,C 180,E1 20814.429,E2 20814.429} C_VEL
LIN {X 0,Y 436.863,Z 1111.165,A -85,B 0,C 180,E1 20811.764,E2 20811.764} C_VEL
LIN {X 0,Y 434.706,Z 1122.525,A -85,B 0,C 180,E1 20808.507,E2 20808.507} C_VEL
LIN {X 0,Y 433.474,Z 1130.382,A -85,B 0,C 180,E1 20805.795,E2 20805.795} C_VEL
LIN {X 0,Y 432.554,Z 1138.078,A -85,B 0,C 180,E1 20802.55,E2 20802.55} C_VEL
LIN {X 0,Y 432.138,Z 1143.265,A -85,B 0,C 180,E1 20799.703,E2 20799.703} C_VEL
LIN {X 0,Y 431.978,Z 1147.113,A -85,B 0,C 180,E1 20796.913,E2 20796.913} C_VEL
LIN {X 0,Y 431.94,Z 1149.892,A -85,B 0,C 180,E1 20793.716,E2 20793.716} C_VEL
LIN {X 0,Y 431.941,Z 1150.918,A -85,B 0,C 180,E1 20791.061,E2 20791.061} C_VEL
LIN {X 0,Y 431.943,Z 1150.846,A -85,B 0,C 180,E1 20788.541,E2 20788.541} C_VEL
LIN {X 0,Y 431.937,Z 1149.273,A -85,B 0,C 180,E1 20785.353,E2 20785.353} C_VEL
LIN {X 0,Y 431.975,Z 1146.441,A -85,B 0,C 180,E1 20782.552,E2 20782.552} C_VEL
LIN {X 0,Y 432.178,Z 1142.578,A -85,B 0,C 180,E1 20779.873,E2 20779.873} C_VEL
LIN {X 0,Y 432.77,Z 1135.997,A -85,B 0,C 180,E1 20776.505,E2 20776.505} C_VEL
LIN {X 0,Y 433.631,Z 1129.266,A -85,B 0,C 180,E1 20773.799,E2 20773.799} C_VEL
LIN {X 0,Y 435.18,Z 1119.916,A -85,B 0,C 180,E1 20770.679,E2 20770.679} C_VEL
LIN {X 0,Y 437.19,Z 1109.551,A -85,B 0,C 180,E1 20767.829,E2 20767.829} C_VEL
LIN {X 0,Y 439.892,Z 1097.566,A -85,B 0,C 180,E1 20764.989,E2 20764.989} C_VEL
LIN {X 0,Y 443.124,Z 1084.105,A -85,B 0,C 180,E1 20762.301,E2 20762.301} C_VEL
LIN {X 0,Y 446.938,Z 1069.296,A -85,B 0,C 180,E1 20759.719,E2 20759.719} C_VEL
LIN {X 0,Y 451.228,Z 1052.755,A -85,B 0,C 180,E1 20757.269,E2 20757.269} C_VEL
LIN {X 0,Y 455.874,Z 1035.212,A -85,B 0,C 180,E1 20755.006,E2 20755.006} C_VEL
LIN {X 0,Y 460.608,Z 1016.515,A -85,B 0,C 180,E1 20752.958,E2 20752.958} C_VEL
LIN {X 0,Y 465.521,Z 996.712,A -85,B 0,C 180,E1 20751.078,E2 20751.078} C_VEL
LIN {X 0,Y 470.108,Z 976.685,A -85,B 0,C 180,E1 20749.475,E2 20749.475} C_VEL
LIN {X 0,Y 474.651,Z 955.592,A -85,B 0,C 180,E1 20748.022,E2 20748.022} C_VEL
LIN {X 0,Y 478.838,Z 933.537,A -85,B 0,C 180,E1 20746.771,E2 20746.771} C_VEL
LIN {X 0,Y 482.383,Z 912.598,A -85,B 0,C 180,E1 20745.772,E2 20745.772} C_VEL
LIN {X 0,Y 485.763,Z 888.9,A -85,B 0,C 180,E1 20744.869,E2 20744.869} C_VEL
LIN {X 0,Y 488.257,Z 867.709,A -85,B 0,C 180,E1 20744.235,E2 20744.235} C_VEL
LIN {X 0,Y 490.475,Z 841.539,A -85,B 0,C 180,E1 20743.657,E2 20743.657} C_VEL
LIN {X 0,Y 500.871,Z 616.939,A -85,B 0,C 180,E1 20740.088,E2 20740.088} C_VEL
LIN {X 0,Y 503.966,Z 548.444,A -85,B 0,C 180,E1 20738.992,E2 20738.992} C_VEL
LIN {X 0,Y 492.935,Z 530.196,A -85,B 0,C 180,E1 20737.064,E2 20737.064} C_VEL
LIN {X 0,Y 481.06,Z 511.999,A -85,B 0,C 180,E1 20734.825,E2 20734.825} C_VEL
LIN {X 0,Y 469.522,Z 495.876,A -85,B 0,C 180,E1 20732.457,E2 20732.457} C_VEL
LIN {X 0,Y 460.023,Z 483.368,A -85,B 0,C 180,E1 20730.319,E2 20730.319} C_VEL
LIN {X 0,Y 454.829,Z 476.922,A -85,B 0,C 180,E1 20729.068,E2 20729.068} C_VEL
LIN {X 0,Y 451.261,Z 472.428,A -85,B 0,C 180,E1 20728.162,E2 20728.162} C_VEL
LIN {X 0,Y 447.032,Z 467.14,A -85,B 0,C 180,E1 20727.004,E2 20727.004} C_VEL
LIN {X 0,Y 444.49,Z 462.32,A -85,B 0,C 180,E1 20725.446,E2 20725.446} C_VEL
LIN {X 0,Y 442.202,Z 457.836,A -85,B 0,C 180,E1 20723.875,E2 20723.875} C_VEL
LIN {X 0,Y 440.19,Z 454.056,A -85,B 0,C 180,E1 20722.434,E2 20722.434} C_VEL
LIN {X 0,Y 437.55,Z 449.415,A -85,B 0,C 180,E1 20720.457,E2 20720.457} C_VEL
LIN {X 0,Y 436.791,Z 447.906,A -85,B 0,C 180,E1 20719.804,E2 20719.804} C_VEL
LIN {X 0,Y 434.715,Z 444.47,A -85,B 0,C 180,E1 20718.09,E2 20718.09} C_VEL
LIN {X 0,Y 434.399,Z 443.233,A -85,B 0,C 180,E1 20717.412,E2 20717.412} C_VEL
LIN {X 0,Y 434.395,Z 443.089,A -85,B 0,C 180,E1 20713.715,E2 20713.715} C_VEL
LIN {X 0,Y 434.411,Z 443.085,A -85,B 0,C 180,E1 20709.941,E2 20709.941} C_VEL
LIN {X 0,Y 434.389,Z 443.095,A -85,B 0,C 180,E1 20706.343,E2 20706.343} C_VEL
LIN {X 0,Y 434.366,Z 443.115,A -85,B 0,C 180,E1 20702.639,E2 20702.639} C_VEL
LIN {X 0,Y 434.36,Z 443.119,A -85,B 0,C 180,E1 20698.945,E2 20698.945} C_VEL
LIN {X 0,Y 434.368,Z 443.097,A -85,B 0,C 180,E1 20695.246,E2 20695.246} C_VEL
LIN {X 0,Y 434.403,Z 443.084,A -85,B 0,C 180,E1 20691.662,E2 20691.662} C_VEL
LIN {X 0,Y 434.378,Z 443.091,A -85,B 0,C 180,E1 20687.909,E2 20687.909} C_VEL
LIN {X 0,Y 434.345,Z 443.107,A -85,B 0,C 180,E1 20684.375,E2 20684.375} C_VEL
LIN {X 0,Y 434.434,Z 443.426,A -85,B 0,C 180,E1 20681.417,E2 20681.417} C_VEL
LIN {X 0,Y 435.815,Z 446.79,A -85,B 0,C 180,E1 20679.87,E2 20679.87} C_VEL
LIN {X 0,Y 437.257,Z 448.784,A -85,B 0,C 180,E1 20678.82,E2 20678.82} C_VEL
LIN {X 0,Y 439.387,Z 452.828,A -85,B 0,C 180,E1 20677.099,E2 20677.099} C_VEL
LIN {X 0,Y 442.63,Z 458.964,A -85,B 0,C 180,E1 20674.726,E2 20674.726} C_VEL
LIN {X 0,Y 445.119,Z 463.896,A -85,B 0,C 180,E1 20673.015,E2 20673.015} C_VEL
LIN {X 0,Y 447.364,Z 468.339,A -85,B 0,C 180,E1 20671.571,E2 20671.571} C_VEL
LIN {X 0,Y 451.49,Z 476.683,A -85,B 0,C 180,E1 20669.083,E2 20669.083} C_VEL
LIN {X 0,Y 455.863,Z 485.907,A -85,B 0,C 180,E1 20666.688,E2 20666.688} C_VEL
LIN {X 0,Y 465.834,Z 499.816,A -85,B 0,C 180,E1 20664.355,E2 20664.355} C_VEL
LIN {X 0,Y 476.083,Z 515.071,A -85,B 0,C 180,E1 20662.173,E2 20662.173} C_VEL
LIN {X 0,Y 487.115,Z 532.43,A -85,B 0,C 180,E1 20660.022,E2 20660.022} C_VEL
LIN {X 0,Y 497.337,Z 550.038,A -85,B 0,C 180,E1 20658.165,E2 20658.165} C_VEL
LIN {X 0,Y 500.269,Z 555.68,A -85,B 0,C 180,E1 20657.647,E2 20657.647} C_VEL
LIN {X 0,Y 501.682,Z 565.791,A -85,B 0,C 180,E1 20657.247,E2 20657.247} C_VEL
LIN {X 0,Y 491.161,Z 822.511,A -85,B 0,C 180,E1 20653.412,E2 20653.412} C_VEL
LIN {X 0,Y 489.501,Z 854.013,A -85,B 0,C 180,E1 20652.89,E2 20652.89} C_VEL
LIN {X 0,Y 487.439,Z 875.789,A -85,B 0,C 180,E1 20652.371,E2 20652.371} C_VEL
LIN {X 0,Y 484.39,Z 899.978,A -85,B 0,C 180,E1 20651.579,E2 20651.579} C_VEL
LIN {X 0,Y 481.113,Z 921.075,A -85,B 0,C 180,E1 20650.694,E2 20650.694} C_VEL
LIN {X 0,Y 477.151,Z 942.5,A -85,B 0,C 180,E1 20649.572,E2 20649.572} C_VEL
LIN {X 0,Y 472.999,Z 962.362,A -85,B 0,C 180,E1 20648.325,E2 20648.325} C_VEL
LIN {X 0,Y 468.301,Z 982.424,A -85,B 0,C 180,E1 20646.805,E2 20646.805} C_VEL
LIN {X 0,Y 463.642,Z 1000.963,A -85,B 0,C 180,E1 20645.157,E2 20645.157} C_VEL
LIN {X 0,Y 458.708,Z 1019.045,A -85,B 0,C 180,E1 20643.245,E2 20643.245} C_VEL
LIN {X 0,Y 454.005,Z 1035.907,A -85,B 0,C 180,E1 20641.169,E2 20641.169} C_VEL
LIN {X 0,Y 449.664,Z 1050.837,A -85,B 0,C 180,E1 20638.997,E2 20638.997} C_VEL
LIN {X 0,Y 445.465,Z 1065.464,A -85,B 0,C 180,E1 20636.531,E2 20636.531} C_VEL
LIN {X 0,Y 441.923,Z 1077.962,A -85,B 0,C 180,E1 20634.033,E2 20634.033} C_VEL
LIN {X 0,Y 438.632,Z 1090.363,A -85,B 0,C 180,E1 20631.111,E2 20631.111} C_VEL
LIN {X 0,Y 436.289,Z 1099.916,A -85,B 0,C 180,E1 20628.412,E2 20628.412} C_VEL
LIN {X 0,Y 434.368,Z 1108.949,A -85,B 0,C 180,E1 20625.308,E2 20625.308} C_VEL
LIN {X 0,Y 433.215,Z 1115.554,A -85,B 0,C 180,E1 20622.494,E2 20622.494} C_VEL
LIN {X 0,Y 432.446,Z 1121.267,A -85,B 0,C 180,E1 20619.314,E2 20619.314} C_VEL
LIN {X 0,Y 432.439,Z 1121.337,A -85,B 0,C 180,E1 20619.268,E2 20619.268} C_VEL
LIN {X 0,Y 431.307,Z 1122.896,A -85,B 0,C 180,E1 20618.268,E2 20618.268} C_VEL
LIN {X 0,Y 424.696,Z 1126.18,A -85,B 0,C 180,E1 20615.515,E2 20615.515} C_VEL
LIN {X 0,Y 424.018,Z 1126.842,A -85,B 0,C 180,E1 20614.697,E2 20614.697} C_VEL
LIN {X 0,Y 423.956,Z 1128.411,A -85,B 0,C 180,E1 20611.487,E2 20611.487} C_VEL
LIN {X 0,Y 423.958,Z 1128.47,A -85,B 0,C 180,E1 20608.784,E2 20608.784} C_VEL
LIN {X 0,Y 424.005,Z 1127.22,A -85,B 0,C 180,E1 20605.672,E2 20605.672} C_VEL
LIN {X 0,Y 424.181,Z 1124.475,A -85,B 0,C 180,E1 20602.687,E2 20602.687} C_VEL
LIN {X 0,Y 424.663,Z 1120.209,A -85,B 0,C 180,E1 20599.554,E2 20599.554} C_VEL
LIN {X 0,Y 425.526,Z 1114.445,A -85,B 0,C 180,E1 20596.548,E2 20596.548} C_VEL
LIN {X 0,Y 426.967,Z 1107.237,A -85,B 0,C 180,E1 20593.539,E2 20593.539} C_VEL
LIN {X 0,Y 429.064,Z 1098.154,A -85,B 0,C 180,E1 20590.534,E2 20590.534} C_VEL
LIN {X 0,Y 431.942,Z 1087.291,A -85,B 0,C 180,E1 20587.545,E2 20587.545} C_VEL
LIN {X 0,Y 435.097,Z 1076.168,A -85,B 0,C 180,E1 20584.985,E2 20584.985} C_VEL
LIN {X 0,Y 439.361,Z 1061.83,A -85,B 0,C 180,E1 20582.19,E2 20582.19} C_VEL
LIN {X 0,Y 443.678,Z 1047.546,A -85,B 0,C 180,E1 20579.83,E2 20579.83} C_VEL
LIN {X 0,Y 448.614,Z 1030.97,A -85,B 0,C 180,E1 20577.51,E2 20577.51} C_VEL
LIN {X 0,Y 453.555,Z 1014.101,A -85,B 0,C 180,E1 20575.488,E2 20575.488} C_VEL
LIN {X 0,Y 458.591,Z 995.633,A -85,B 0,C 180,E1 20573.626,E2 20573.626} C_VEL
LIN {X 0,Y 463.507,Z 976.609,A -85,B 0,C 180,E1 20571.983,E2 20571.983} C_VEL
LIN {X 0,Y 468.076,Z 956.906,A -85,B 0,C 180,E1 20570.569,E2 20570.569} C_VEL
LIN {X 0,Y 472.459,Z 936.232,A -85,B 0,C 180,E1 20569.319,E2 20569.319} C_VEL
LIN {X 0,Y 476.126,Z 915.844,A -85,B 0,C 180,E1 20568.315,E2 20568.315} C_VEL
LIN {X 0,Y 479.635,Z 893.301,A -85,B 0,C 180,E1 20567.415,E2 20567.415} C_VEL
LIN {X 0,Y 482.247,Z 871.557,A -85,B 0,C 180,E1 20566.754,E2 20566.754} C_VEL
LIN {X 0,Y 484.391,Z 847.722,A -85,B 0,C 180,E1 20566.221,E2 20566.221} C_VEL
LIN {X 0,Y 488.222,Z 758.983,A -85,B 0,C 180,E1 20564.864,E2 20564.864} C_VEL
LIN {X 0,Y 496.422,Z 566.016,A -85,B 0,C 180,E1 20561.939,E2 20561.939} C_VEL
LIN {X 0,Y 495.23,Z 559.122,A -85,B 0,C 180,E1 20561.626,E2 20561.626} C_VEL
LIN {X 0,Y 484.628,Z 540.56,A -85,B 0,C 180,E1 20559.672,E2 20559.672} C_VEL
LIN {X 0,Y 474.391,Z 524.009,A -85,B 0,C 180,E1 20557.642,E2 20557.642} C_VEL
LIN {X 0,Y 465.777,Z 510.923,A -85,B 0,C 180,E1 20555.802,E2 20555.802} C_VEL
LIN {X 0,Y 456.378,Z 497.492,A -85,B 0,C 180,E1 20553.625,E2 20553.625} C_VEL
LIN {X 0,Y 451.039,Z 490.217,A -85,B 0,C 180,E1 20552.294,E2 20552.294} C_VEL
LIN {X 0,Y 446.873,Z 484.313,A -85,B 0,C 180,E1 20551.123,E2 20551.123} C_VEL
LIN {X 0,Y 443.177,Z 476.611,A -85,B 0,C 180,E1 20548.87,E2 20548.87} C_VEL
LIN {X 0,Y 440.916,Z 472.044,A -85,B 0,C 180,E1 20547.41,E2 20547.41} C_VEL
LIN {X 0,Y 438.995,Z 468.075,A -85,B 0,C 180,E1 20546.078,E2 20546.078} C_VEL
LIN {X 0,Y 436.569,Z 463.359,A -85,B 0,C 180,E1 20544.347,E2 20544.347} C_VEL
LIN {X 0,Y 434.126,Z 458.704,A -85,B 0,C 180,E1 20542.479,E2 20542.479} C_VEL
LIN {X 0,Y 432.198,Z 454.85,A -85,B 0,C 180,E1 20540.827,E2 20540.827} C_VEL
LIN {X 0,Y 429.624,Z 450.445,A -85,B 0,C 180,E1 20538.593,E2 20538.593} C_VEL
LIN {X 0,Y 428.815,Z 448.92,A -85,B 0,C 180,E1 20537.786,E2 20537.786} C_VEL
LIN {X 0,Y 426.495,Z 444.692,A -85,B 0,C 180,E1 20535.223,E2 20535.223} C_VEL
LIN {X 0,Y 426.469,Z 444.14,A -85,B 0,C 180,E1 20534.39,E2 20534.39} C_VEL
LIN {X 0,Y 426.444,Z 444.108,A -85,B 0,C 180,E1 20530.538,E2 20530.538} C_VEL
LIN {X 0,Y 426.417,Z 444.091,A -85,B 0,C 180,E1 20526.868,E2 20526.868} C_VEL
LIN {X 0,Y 426.41,Z 444.081,A -85,B 0,C 180,E1 20523.092,E2 20523.092} C_VEL
LIN {X 0,Y 426.417,Z 444.078,A -85,B 0,C 180,E1 20519.328,E2 20519.328} C_VEL
LIN {X 0,Y 426.434,Z 444.085,A -85,B 0,C 180,E1 20515.562,E2 20515.562} C_VEL
LIN {X 0,Y 426.476,Z 444.098,A -85,B 0,C 180,E1 20511.913,E2 20511.913} C_VEL
LIN {X 0,Y 426.477,Z 444.109,A -85,B 0,C 180,E1 20507.956,E2 20507.956} C_VEL
LIN {X 0,Y 426.531,Z 444.457,A -85,B 0,C 180,E1 20505.732,E2 20505.732} C_VEL
LIN {X 0,Y 428.231,Z 448.201,A -85,B 0,C 180,E1 20503.589,E2 20503.589} C_VEL
LIN {X 0,Y 429.618,Z 450.184,A -85,B 0,C 180,E1 20502.388,E2 20502.388} C_VEL
LIN {X 0,Y 431.689,Z 453.987,A -85,B 0,C 180,E1 20500.512,E2 20500.512} C_VEL
LIN {X 0,Y 432.528,Z 455.491,A -85,B 0,C 180,E1 20499.813,E2 20499.813} C_VEL
LIN {X 0,Y 434.507,Z 459.05,A -85,B 0,C 180,E1 20498.254,E2 20498.254} C_VEL
LIN {X 0,Y 437.739,Z 465.211,A -85,B 0,C 180,E1 20495.866,E2 20495.866} C_VEL
LIN {X 0,Y 439.43,Z 468.328,A -85,B 0,C 180,E1 20494.853,E2 20494.853} C_VEL
LIN {X 0,Y 446.189,Z 476.482,A -85,B 0,C 180,E1 20492.904,E2 20492.904} C_VEL
LIN {X 0,Y 450.857,Z 482.243,A -85,B 0,C 180,E1 20491.667,E2 20491.667} C_VEL
LIN {X 0,Y 455.683,Z 488.41,A -85,B 0,C 180,E1 20490.451,E2 20490.451} C_VEL
LIN {X 0,Y 463.071,Z 497.899,A -85,B 0,C 180,E1 20488.714,E2 20488.714} C_VEL
LIN {X 0,Y 473.11,Z 511.985,A -85,B 0,C 180,E1 20486.522,E2 20486.522} C_VEL
LIN {X 0,Y 483.068,Z 526.641,A -85,B 0,C 180,E1 20484.525,E2 20484.525} C_VEL
LIN {X 0,Y 495.447,Z 546.505,A -85,B 0,C 180,E1 20482.229,E2 20482.229} C_VEL
LIN {X 0,Y 498.804,Z 552.613,A -85,B 0,C 180,E1 20481.627,E2 20481.627} C_VEL
LIN {X 0,Y 487.654,Z 784.908,A -85,B 0,C 180,E1 20477.94,E2 20477.94} C_VEL
LIN {X 0,Y 484.615,Z 845.959,A -85,B 0,C 180,E1 20476.939,E2 20476.939} C_VEL
LIN {X 0,Y 482.265,Z 870.584,A -85,B 0,C 180,E1 20476.36,E2 20476.36} C_VEL
LIN {X 0,Y 479.467,Z 893.214,A -85,B 0,C 180,E1 20475.657,E2 20475.657} C_VEL
LIN {X 0,Y 475.928,Z 916.157,A -85,B 0,C 180,E1 20474.734,E2 20474.734} C_VEL
LIN {X 0,Y 472.315,Z 936.644,A -85,B 0,C 180,E1 20473.726,E2 20473.726} C_VEL
LIN {X 0,Y 467.587,Z 959.877,A -85,B 0,C 180,E1 20472.346,E2 20472.346} C_VEL
LIN {X 0,Y 463.346,Z 978.904,A -85,B 0,C 180,E1 20470.998,E2 20470.998} C_VEL
LIN {X 0,Y 457.919,Z 1001.276,A -85,B 0,C 180,E1 20469.128,E2 20469.128} C_VEL
LIN {X 0,Y 453.259,Z 1019.384,A -85,B 0,C 180,E1 20467.348,E2 20467.348} C_VEL
LIN {X 0,Y 447.966,Z 1039.107,A -85,B 0,C 180,E1 20465.083,E2 20465.083} C_VEL
LIN {X 0,Y 443.637,Z 1054.899,A -85,B 0,C 180,E1 20462.977,E2 20462.977} C_VEL
LIN {X 0,Y 438.927,Z 1072.16,A -85,B 0,C 180,E1 20460.302,E2 20460.302} C_VEL
LIN {X 0,Y 435.42,Z 1085.325,A -85,B 0,C 180,E1 20457.935,E2 20457.935} C_VEL
LIN {X 0,Y 431.787,Z 1099.719,A -85,B 0,C 180,E1 20454.927,E2 20454.927} C_VEL
LIN {X 0,Y 429.303,Z 1110.393,A -85,B 0,C 180,E1 20452.312,E2 20452.312} C_VEL
LIN {X 0,Y 427.064,Z 1121.456,A -85,B 0,C 180,E1 20449.134,E2 20449.134} C_VEL
LIN {X 0,Y 425.644,Z 1129.789,A -85,B 0,C 180,E1 20446.233,E2 20446.233} C_VEL
LIN {X 0,Y 424.666,Z 1137.33,A -85,B 0,C 180,E1 20443.064,E2 20443.064} C_VEL
LIN {X 0,Y 424.17,Z 1142.8,A -85,B 0,C 180,E1 20440.046,E2 20440.046} C_VEL
LIN {X 0,Y 423.976,Z 1146.567,A -85,B 0,C 180,E1 20437.317,E2 20437.317} C_VEL
LIN {X 0,Y 423.944,Z 1149.467,A -85,B 0,C 180,E1 20434.193,E2 20434.193} C_VEL
LIN {X 0,Y 423.947,Z 1150.661,A -85,B 0,C 180,E1 20431.351,E2 20431.351} C_VEL
LIN {X 0,Y 423.947,Z 1150.683,A -85,B 0,C 180,E1 20428.784,E2 20428.784} C_VEL
LIN {X 0,Y 423.942,Z 1149.535,A -85,B 0,C 180,E1 20425.943,E2 20425.943} C_VEL
LIN {X 0,Y 423.98,Z 1146.724,A -85,B 0,C 180,E1 20422.82,E2 20422.82} C_VEL
LIN {X 0,Y 424.157,Z 1143.004,A -85,B 0,C 180,E1 20420.091,E2 20420.091} C_VEL
LIN {X 0,Y 424.635,Z 1137.58,A -85,B 0,C 180,E1 20417.074,E2 20417.074} C_VEL
LIN {X 0,Y 425.588,Z 1130.131,A -85,B 0,C 180,E1 20413.905,E2 20413.905} C_VEL
LIN {X 0,Y 426.98,Z 1121.85,A -85,B 0,C 180,E1 20411.004,E2 20411.004} C_VEL
LIN {X 0,Y 429.185,Z 1110.894,A -85,B 0,C 180,E1 20407.826,E2 20407.826} C_VEL
LIN {X 0,Y 431.639,Z 1100.274,A -85,B 0,C 180,E1 20405.21,E2 20405.21} C_VEL
LIN {X 0,Y 435.255,Z 1085.9,A -85,B 0,C 180,E1 20402.183,E2 20402.183} C_VEL
LIN {X 0,Y 438.912,Z 1072.122,A -85,B 0,C 180,E1 20399.701,E2 20399.701} C_VEL
LIN {X 0,Y 443.755,Z 1054.35,A -85,B 0,C 180,E1 20396.956,E2 20396.956} C_VEL
LIN {X 0,Y 448.099,Z 1038.503,A -85,B 0,C 180,E1 20394.851,E2 20394.851} C_VEL
LIN {X 0,Y 453.415,Z 1018.589,A -85,B 0,C 180,E1 20392.58,E2 20392.58} C_VEL
LIN {X 0,Y 457.902,Z 1001.143,A -85,B 0,C 180,E1 20390.871,E2 20390.871} C_VEL
LIN {X 0,Y 463.329,Z 978.738,A -85,B 0,C 180,E1 20389,E2 20389} C_VEL
LIN {X 0,Y 467.568,Z 959.697,A -85,B 0,C 180,E1 20387.652,E2 20387.652} C_VEL
LIN {X 0,Y 472.294,Z 936.414,A -85,B 0,C 180,E1 20386.272,E2 20386.272} C_VEL
LIN {X 0,Y 475.908,Z 915.886,A -85,B 0,C 180,E1 20385.264,E2 20385.264} C_VEL
LIN {X 0,Y 479.699,Z 890.902,A -85,B 0,C 180,E1 20384.275,E2 20384.275} C_VEL
LIN {X 0,Y 482.308,Z 869.588,A -85,B 0,C 180,E1 20383.622,E2 20383.622} C_VEL
LIN {X 0,Y 484.64,Z 844.269,A -85,B 0,C 180,E1 20383.04,E2 20383.04} C_VEL
LIN {X 0,Y 489.17,Z 750.469,A -85,B 0,C 180,E1 20381.519,E2 20381.519} C_VEL
LIN {X 0,Y 498.667,Z 552.191,A -85,B 0,C 180,E1 20378.367,E2 20378.367} C_VEL
LIN {X 0,Y 487.787,Z 534.092,A -85,B 0,C 180,E1 20376.401,E2 20376.401} C_VEL
LIN {X 0,Y 476.928,Z 517.483,A -85,B 0,C 180,E1 20374.294,E2 20374.294} C_VEL
LIN {X 0,Y 466.062,Z 502.094,A -85,B 0,C 180,E1 20372,E2 20372} C_VEL
LIN {X 0,Y 456.925,Z 489.964,A -85,B 0,C 180,E1 20369.893,E2 20369.893} C_VEL
LIN {X 0,Y 452.033,Z 483.782,A -85,B 0,C 180,E1 20368.686,E2 20368.686} C_VEL
LIN {X 0,Y 448.399,Z 479.205,A -85,B 0,C 180,E1 20367.742,E2 20367.742} C_VEL
LIN {X 0,Y 443.911,Z 473.735,A -85,B 0,C 180,E1 20366.523,E2 20366.523} C_VEL
LIN {X 0,Y 439.001,Z 467.809,A -85,B 0,C 180,E1 20365.065,E2 20365.065} C_VEL
LIN {X 0,Y 437.101,Z 463.931,A -85,B 0,C 180,E1 20363.742,E2 20363.742} C_VEL
LIN {X 0,Y 435.11,Z 460.16,A -85,B 0,C 180,E1 20362.283,E2 20362.283} C_VEL
LIN {X 0,Y 432.414,Z 455.125,A -85,B 0,C 180,E1 20360.146,E2 20360.146} C_VEL
LIN {X 0,Y 429.748,Z 450.553,A -85,B 0,C 180,E1 20357.886,E2 20357.886} C_VEL
LIN {X 0,Y 428.748,Z 448.811,A -85,B 0,C 180,E1 20356.949,E2 20356.949} C_VEL
LIN {X 0,Y 426.602,Z 444.956,A -85,B 0,C 180,E1 20354.663,E2 20354.663} C_VEL
LIN {X 0,Y 426.486,Z 444.144,A -85,B 0,C 180,E1 20353.974,E2 20353.974} C_VEL
LIN {X 0,Y 426.468,Z 444.074,A -85,B 0,C 180,E1 20350.128,E2 20350.128} C_VEL
LIN {X 0,Y 426.441,Z 444.085,A -85,B 0,C 180,E1 20346.462,E2 20346.462} C_VEL
LIN {X 0,Y 426.425,Z 444.104,A -85,B 0,C 180,E1 20342.688,E2 20342.688} C_VEL
LIN {X 0,Y 426.421,Z 444.107,A -85,B 0,C 180,E1 20338.925,E2 20338.925} C_VEL
LIN {X 0,Y 426.424,Z 444.087,A -85,B 0,C 180,E1 20335.158,E2 20335.158} C_VEL
LIN {X 0,Y 426.452,Z 444.074,A -85,B 0,C 180,E1 20331.505,E2 20331.505} C_VEL
LIN {X 0,Y 426.454,Z 444.076,A -85,B 0,C 180,E1 20327.68,E2 20327.68} C_VEL
LIN {X 0,Y 426.439,Z 444.325,A -85,B 0,C 180,E1 20324.775,E2 20324.775} C_VEL
LIN {X 0,Y 428.561,Z 448.628,A -85,B 0,C 180,E1 20322.203,E2 20322.203} C_VEL
LIN {X 0,Y 429.519,Z 450.107,A -85,B 0,C 180,E1 20321.347,E2 20321.347} C_VEL
LIN {X 0,Y 431.316,Z 453.578,A -85,B 0,C 180,E1 20319.651,E2 20319.651} C_VEL
LIN {X 0,Y 432.302,Z 455.23,A -85,B 0,C 180,E1 20318.849,E2 20318.849} C_VEL
LIN {X 0,Y 434.962,Z 460.219,A -85,B 0,C 180,E1 20316.709,E2 20316.709} C_VEL
LIN {X 0,Y 437.473,Z 465.081,A -85,B 0,C 180,E1 20314.837,E2 20314.837} C_VEL
LIN {X 0,Y 439.927,Z 470.012,A -85,B 0,C 180,E1 20313.109,E2 20313.109} C_VEL
LIN {X 0,Y 442.322,Z 474.94,A -85,B 0,C 180,E1 20311.512,E2 20311.512} C_VEL
LIN {X 0,Y 446.02,Z 482.363,A -85,B 0,C 180,E1 20309.261,E2 20309.261} C_VEL
LIN {X 0,Y 447.887,Z 485.828,A -85,B 0,C 180,E1 20308.394,E2 20308.394} C_VEL
LIN {X 0,Y 458.538,Z 500.431,A -85,B 0,C 180,E1 20305.726,E2 20305.726} C_VEL
LIN {X 0,Y 470.945,Z 518.628,A -85,B 0,C 180,E1 20302.955,E2 20302.955} C_VEL
LIN {X 0,Y 483.138,Z 538.099,A -85,B 0,C 180,E1 20300.495,E2 20300.495} C_VEL
LIN {X 0,Y 493.465,Z 556.125,A -85,B 0,C 180,E1 20298.572,E2 20298.572} C_VEL
LIN {X 0,Y 495.435,Z 560.107,A -85,B 0,C 180,E1 20298.211,E2 20298.211} C_VEL
LIN {X 0,Y 496.388,Z 567.55,A -85,B 0,C 180,E1 20297.92,E2 20297.92} C_VEL
LIN {X 0,Y 485.488,Z 823.755,A -85,B 0,C 180,E1 20294.063,E2 20294.063} C_VEL
LIN {X 0,Y 483.757,Z 854.76,A -85,B 0,C 180,E1 20293.541,E2 20293.541} C_VEL
LIN {X 0,Y 481.611,Z 876.638,A -85,B 0,C 180,E1 20293.011,E2 20293.011} C_VEL
LIN {X 0,Y 478.565,Z 899.931,A -85,B 0,C 180,E1 20292.241,E2 20292.241} C_VEL
LIN {X 0,Y 475.199,Z 920.974,A -85,B 0,C 180,E1 20291.354,E2 20291.354} C_VEL
LIN {X 0,Y 471.002,Z 942.98,A -85,B 0,C 180,E1 20290.193,E2 20290.193} C_VEL
LIN {X 0,Y 466.591,Z 963.414,A -85,B 0,C 180,E1 20288.895,E2 20288.895} C_VEL
LIN {X 0,Y 461.795,Z 983.099,A -85,B 0,C 180,E1 20287.379,E2 20287.379} C_VEL
LIN {X 0,Y 456.889,Z 1001.95,A -85,B 0,C 180,E1 20285.678,E2 20285.678} C_VEL
LIN {X 0,Y 451.794,Z 1019.902,A -85,B 0,C 180,E1 20283.745,E2 20283.745} C_VEL
LIN {X 0,Y 446.784,Z 1037.099,A -85,B 0,C 180,E1 20281.58,E2 20281.58} C_VEL
LIN {X 0,Y 442.311,Z 1051.939,A -85,B 0,C 180,E1 20279.377,E2 20279.377} C_VEL
LIN {X 0,Y 437.739,Z 1067.149,A -85,B 0,C 180,E1 20276.73,E2 20276.73} C_VEL
LIN {X 0,Y 434.133,Z 1079.452,A -85,B 0,C 180,E1 20274.203,E2 20274.203} C_VEL
LIN {X 0,Y 430.889,Z 1091.102,A -85,B 0,C 180,E1 20271.366,E2 20271.366} C_VEL
LIN {X 0,Y 428.479,Z 1100.512,A -85,B 0,C 180,E1 20268.645,E2 20268.645} C_VEL
LIN {X 0,Y 426.481,Z 1109.41,A -85,B 0,C 180,E1 20265.502,E2 20265.502} C_VEL
LIN {X 0,Y 425.23,Z 1116.283,A -85,B 0,C 180,E1 20262.494,E2 20262.494} C_VEL
LIN {X 0,Y 424.462,Z 1121.682,A -85,B 0,C 180,E1 20259.354,E2 20259.354} C_VEL
LIN {X 0,Y 424.117,Z 1125.438,A -85,B 0,C 180,E1 20256.362,E2 20256.362} C_VEL
LIN {X 0,Y 424.018,Z 1126.842,A -85,B 0,C 180,E1 20254.697,E2 20254.697} C_VEL
LIN {X 0,Y 423.004,Z 1127.618,A -85,B 0,C 180,E1 20253.662,E2 20253.662} C_VEL
LIN {X 0,Y 418.214,Z 1128.633,A -85,B 0,C 180,E1 20251.631,E2 20251.631} C_VEL
LIN {X 0,Y 416.131,Z 1128.858,A -85,B 0,C 180,E1 20250.354,E2 20250.354} C_VEL
LIN {X 0,Y 415.97,Z 1128.859,A -85,B 0,C 180,E1 20249.97,E2 20249.97} C_VEL
LIN {X 0,Y 415.979,Z 1128.059,A -85,B 0,C 180,E1 20246.831,E2 20246.831} C_VEL
LIN {X 0,Y 416.105,Z 1126.014,A -85,B 0,C 180,E1 20243.792,E2 20243.792} C_VEL
LIN {X 0,Y 416.461,Z 1122.24,A -85,B 0,C 180,E1 20240.604,E2 20240.604} C_VEL
LIN {X 0,Y 417.2,Z 1117.237,A -85,B 0,C 180,E1 20237.543,E2 20237.543} C_VEL
LIN {X 0,Y 418.463,Z 1110.565,A -85,B 0,C 180,E1 20234.477,E2 20234.477} C_VEL
LIN {X 0,Y 420.389,Z 1102.354,A -85,B 0,C 180,E1 20231.415,E2 20231.415} C_VEL
LIN {X 0,Y 423.071,Z 1092.187,A -85,B 0,C 180,E1 20228.365,E2 20228.365} C_VEL
LIN {X 0,Y 426.42,Z 1080.749,A -85,B 0,C 180,E1 20225.478,E2 20225.478} C_VEL
LIN {X 0,Y 430.149,Z 1068.504,A -85,B 0,C 180,E1 20222.896,E2 20222.896} C_VEL
LIN {X 0,Y 434.588,Z 1054.439,A -85,B 0,C 180,E1 20220.352,E2 20220.352} C_VEL
LIN {X 0,Y 439.143,Z 1039.819,A -85,B 0,C 180,E1 20218.113,E2 20218.113} C_VEL
LIN {X 0,Y 444.429,Z 1022.592,A -85,B 0,C 180,E1 20215.852,E2 20215.852} C_VEL
LIN {X 0,Y 449.357,Z 1005.78,A -85,B 0,C 180,E1 20213.983,E2 20213.983} C_VEL
LIN {X 0,Y 454.848,Z 985.907,A -85,B 0,C 180,E1 20212.11,E2 20212.11} C_VEL
LIN {X 0,Y 459.348,Z 968.17,A -85,B 0,C 180,E1 20210.696,E2 20210.696} C_VEL
LIN {X 0,Y 464.438,Z 946.046,A -85,B 0,C 180,E1 20209.223,E2 20209.223} C_VEL
LIN {X 0,Y 468.425,Z 926.323,A -85,B 0,C 180,E1 20208.136,E2 20208.136} C_VEL
LIN {X 0,Y 472.267,Z 903.97,A -85,B 0,C 180,E1 20207.14,E2 20207.14} C_VEL
LIN {X 0,Y 475.285,Z 882.789,A -85,B 0,C 180,E1 20206.393,E2 20206.393} C_VEL
LIN {X 0,Y 477.859,Z 858.947,A -85,B 0,C 180,E1 20205.768,E2 20205.768} C_VEL
LIN {X 0,Y 479.508,Z 835.648,A -85,B 0,C 180,E1 20205.332,E2 20205.332} C_VEL
LIN {X 0,Y 490.631,Z 582.767,A -85,B 0,C 180,E1 20201.497,E2 20201.497} C_VEL
LIN {X 0,Y 491.199,Z 567.606,A -85,B 0,C 180,E1 20201.246,E2 20201.246} C_VEL
LIN {X 0,Y 490.454,Z 563.558,A -85,B 0,C 180,E1 20201.05,E2 20201.05} C_VEL
LIN {X 0,Y 480.061,Z 545.192,A -85,B 0,C 180,E1 20199.074,E2 20199.074} C_VEL
LIN {X 0,Y 470.255,Z 529.282,A -85,B 0,C 180,E1 20197.071,E2 20197.071} C_VEL
LIN {X 0,Y 462.146,Z 516.802,A -85,B 0,C 180,E1 20195.288,E2 20195.288} C_VEL
LIN {X 0,Y 453.245,Z 503.922,A -85,B 0,C 180,E1 20193.169,E2 20193.169} C_VEL
LIN {X 0,Y 448.206,Z 496.975,A -85,B 0,C 180,E1 20191.881,E2 20191.881} C_VEL
LIN {X 0,Y 441.266,Z 487.674,A -85,B 0,C 180,E1 20189.977,E2 20189.977} C_VEL
LIN {X 0,Y 438.477,Z 483.47,A -85,B 0,C 180,E1 20189.06,E2 20189.06} C_VEL
LIN {X 0,Y 433.848,Z 474.143,A -85,B 0,C 180,E1 20185.97,E2 20185.97} C_VEL
LIN {X 0,Y 431.24,Z 469.131,A -85,B 0,C 180,E1 20184.084,E2 20184.084} C_VEL
LIN {X 0,Y 429.031,Z 464.788,A -85,B 0,C 180,E1 20182.327,E2 20182.327} C_VEL
LIN {X 0,Y 426.699,Z 460.215,A -85,B 0,C 180,E1 20180.292,E2 20180.292} C_VEL
LIN {X 0,Y 424.72,Z 456.844,A -85,B 0,C 180,E1 20178.531,E2 20178.531} C_VEL
LIN {X 0,Y 423.96,Z 455.259,A -85,B 0,C 180,E1 20177.713,E2 20177.713} C_VEL
LIN {X 0,Y 421.54,Z 450.733,A -85,B 0,C 180,E1 20174.984,E2 20174.984} C_VEL
LIN {X 0,Y 418.53,Z 445.228,A -85,B 0,C 180,E1 20170.392,E2 20170.392} C_VEL
LIN {X 0,Y 418.499,Z 445.082,A -85,B 0,C 180,E1 20166.585,E2 20166.585} C_VEL
LIN {X 0,Y 418.478,Z 445.07,A -85,B 0,C 180,E1 20162.861,E2 20162.861} C_VEL
LIN {X 0,Y 418.476,Z 445.067,A -85,B 0,C 180,E1 20159.179,E2 20159.179} C_VEL
LIN {X 0,Y 418.484,Z 445.071,A -85,B 0,C 180,E1 20155.34,E2 20155.34} C_VEL
LIN {X 0,Y 418.512,Z 445.087,A -85,B 0,C 180,E1 20151.62,E2 20151.62} C_VEL
LIN {X 0,Y 418.597,Z 445.526,A -85,B 0,C 180,E1 20150.097,E2 20150.097} C_VEL
LIN {X 0,Y 420.957,Z 449.936,A -85,B 0,C 180,E1 20146.539,E2 20146.539} C_VEL
LIN {X 0,Y 421.777,Z 451.3,A -85,B 0,C 180,E1 20145.586,E2 20145.586} C_VEL
LIN {X 0,Y 424.077,Z 455.323,A -85,B 0,C 180,E1 20143.141,E2 20143.141} C_VEL
LIN {X 0,Y 424.974,Z 457.196,A -85,B 0,C 180,E1 20142.19,E2 20142.19} C_VEL
LIN {X 0,Y 427.477,Z 461.473,A -85,B 0,C 180,E1 20140.032,E2 20140.032} C_VEL
LIN {X 0,Y 429.434,Z 465.164,A -85,B 0,C 180,E1 20138.415,E2 20138.415} C_VEL
LIN {X 0,Y 431.468,Z 469.09,A -85,B 0,C 180,E1 20136.979,E2 20136.979} C_VEL
LIN {X 0,Y 434.43,Z 472.566,A -85,B 0,C 180,E1 20135.995,E2 20135.995} C_VEL
LIN {X 0,Y 439.066,Z 478.019,A -85,B 0,C 180,E1 20134.578,E2 20134.578} C_VEL
LIN {X 0,Y 443.708,Z 483.633,A -85,B 0,C 180,E1 20133.248,E2 20133.248} C_VEL
LIN {X 0,Y 448.428,Z 489.543,A -85,B 0,C 180,E1 20131.971,E2 20131.971} C_VEL
LIN {X 0,Y 456.186,Z 499.485,A -85,B 0,C 180,E1 20130.017,E2 20130.017} C_VEL
LIN {X 0,Y 466.147,Z 513.197,A -85,B 0,C 180,E1 20127.716,E2 20127.716} C_VEL
LIN {X 0,Y 477.041,Z 529.13,A -85,B 0,C 180,E1 20125.424,E2 20125.424} C_VEL
LIN {X 0,Y 489.57,Z 549.188,A -85,B 0,C 180,E1 20123.005,E2 20123.005} C_VEL
LIN {X 0,Y 493.48,Z 556.275,A -85,B 0,C 180,E1 20122.281,E2 20122.281} C_VEL
LIN {X 0,Y 482.026,Z 787.414,A -85,B 0,C 180,E1 20118.588,E2 20118.588} C_VEL
LIN {X 0,Y 478.99,Z 846.272,A -85,B 0,C 180,E1 20117.615,E2 20117.615} C_VEL
LIN {X 0,Y 476.59,Z 870.681,A -85,B 0,C 180,E1 20117.036,E2 20117.036} C_VEL
LIN {X 0,Y 473.728,Z 893.187,A -85,B 0,C 180,E1 20116.334,E2 20116.334} C_VEL
LIN {X 0,Y 469.977,Z 916.73,A -85,B 0,C 180,E1 20115.379,E2 20115.379} C_VEL
